Yaskawa INFORM job: DPRINT3D9.JBI

/JOB
//NAME DPRINT3D9
//POS
///NPOS 990,0,0,0,0,0
///TOOL 9
///POSTYPE PULSE
///PULSE
C00000=28405,51687,-122249,62656,-119296,-93988,0
C00001=28412,51716,-122153,62661,-119336,-93961,0
C00002=28422,51752,-122032,62666,-119387,-93929,0
C00003=28439,51788,-121908,62666,-119441,-93896,0
C00004=28474,51840,-121733,62650,-119521,-93851,0
C00005=28491,51862,-121660,62641,-119556,-93833,0
C00006=28516,51888,-121571,62626,-119598,-93812,0
C00007=28569,51934,-121420,62588,-119677,-93776,0
C00008=28598,51956,-121347,62567,-119716,-93759,0
C00009=28631,51978,-121273,62542,-119756,-93743,0
C00010=28686,52010,-121168,62495,-119817,-93721,0
C00011=28702,52019,-121138,62481,-119834,-93715,0
C00012=28783,52055,-121016,62410,-119911,-93692,0
C00013=28872,52087,-120913,62327,-119983,-93676,0
C00014=28965,52116,-120819,62238,-120053,-93663,0
C00015=29065,52138,-120745,62139,-120119,-93656,0
C00016=29167,52158,-120681,62036,-120181,-93653,0
C00017=29273,52171,-120639,61925,-120237,-93656,0
C00018=29381,52181,-120608,61811,-120288,-93663,0
C00019=29407,52182,-120605,61783,-120299,-93666,0
C00020=29496,52184,-120600,61686,-120334,-93678,0
C00021=29604,52182,-120611,61566,-120368,-93696,0
C00022=29681,52175,-120634,61479,-120388,-93714,0
C00023=29759,52166,-120666,61388,-120404,-93733,0
C00024=29816,52159,-120690,61322,-120414,-93748,0
C00025=29867,52150,-120721,61262,-120421,-93765,0
C00026=29912,52141,-120753,61208,-120425,-93780,0
C00027=30014,52117,-120835,61084,-120429,-93818,0
C00028=30081,52097,-120903,61002,-120426,-93846,0
C00029=30142,52075,-120975,60925,-120419,-93875,0
C00030=30190,52057,-121036,60863,-120412,-93899,0
C00031=30233,52039,-121099,60807,-120402,-93923,0
C00032=30261,52025,-121146,60769,-120394,-93940,0
C00033=30336,51984,-121284,60667,-120365,-93989,0
C00034=30393,51946,-121414,60587,-120333,-94033,0
C00035=30394,51945,-121416,60586,-120332,-94033,0
C00036=30454,51900,-121569,60498,-120291,-94084,0
C00037=25336,55338,-110610,67670,-122156,-90253,0
C00038=36363,52336,-120236,76454,-115258,-91971,0
C00039=39662,59274,-99499,75865,-122176,-86210,0
C00040=39594,59234,-99609,75915,-122109,-86232,0
C00041=39523,59198,-99708,75970,-122044,-86250,0
C00042=39446,59171,-99784,76034,-121979,-86261,0
C00043=39368,59147,-99848,76102,-121917,-86268,0
C00044=39340,59142,-99863,76127,-121898,-86268,0
C00045=39232,59125,-99908,76227,-121823,-86266,0
C00046=39175,59121,-99918,76282,-121786,-86261,0
C00047=39120,59120,-99919,76336,-121754,-86254,0
C00048=39037,59123,-99909,76421,-121707,-86239,0
C00049=38943,59135,-99873,76519,-121660,-86216,0
C00050=38887,59145,-99844,76580,-121634,-86200,0
C00051=38833,59159,-99805,76639,-121611,-86181,0
C00052=38779,59174,-99762,76699,-121589,-86161,0
C00053=38727,59193,-99708,76759,-121570,-86138,0
C00054=38679,59214,-99647,76815,-121557,-86114,0
C00055=38626,59240,-99574,76879,-121543,-86085,0
C00056=38582,59266,-99502,76934,-121534,-86059,0
C00057=38541,59294,-99421,76987,-121528,-86030,0
C00058=38493,59330,-99320,77050,-121522,-85994,0
C00059=38457,59362,-99230,77099,-121522,-85963,0
C00060=38425,59397,-99134,77146,-121524,-85931,0
C00061=38384,59443,-99005,77206,-121530,-85888,0
C00062=38358,59479,-98903,77248,-121537,-85855,0
C00063=38335,59518,-98796,77287,-121548,-85821,0
C00064=38305,59573,-98641,77340,-121566,-85773,0
C00065=38288,59612,-98533,77374,-121581,-85739,0
C00066=38275,59653,-98419,77404,-121599,-85704,0
C00067=38258,59716,-98245,77448,-121629,-85652,0
C00068=38251,59756,-98134,77472,-121650,-85619,0
C00069=38248,59798,-98018,77493,-121674,-85585,0
C00070=38246,59850,-97873,77518,-121706,-85543,0
C00071=38249,59905,-97721,77539,-121742,-85499,0
C00072=38262,59984,-97504,77560,-121800,-85439,0
C00073=38270,60017,-97413,77567,-121825,-85414,0
C00074=38282,60058,-97301,77572,-121858,-85383,0
C00075=38312,60130,-97103,77574,-121921,-85331,0
C00076=38328,60164,-97010,77573,-121953,-85306,0
C00077=38348,60200,-96910,77569,-121987,-85280,0
C00078=38384,60252,-96769,77557,-122041,-85245,0
C00079=38395,60266,-96729,77553,-122058,-85235,0
C00080=38449,60329,-96560,77528,-122129,-85194,0
C00081=38511,60384,-96409,77490,-122202,-85159,0
C00082=38578,60436,-96267,77449,-122276,-85127,0
C00083=38651,60480,-96148,77396,-122349,-85104,0
C00084=38728,60520,-96039,77339,-122421,-85083,0
C00085=38809,60551,-95956,77273,-122491,-85071,0
C00086=38893,60578,-95885,77204,-122560,-85063,0
C00087=38913,60582,-95874,77186,-122575,-85062,0
C00088=38984,60595,-95840,77122,-122628,-85063,0
C00089=39071,60603,-95818,77042,-122686,-85069,0
C00090=39134,60603,-95821,76980,-122725,-85079,0
C00091=39199,60598,-95835,76914,-122762,-85093,0
C00092=39246,60594,-95846,76866,-122790,-85102,0
C00093=39289,60587,-95867,76821,-122811,-85115,0
C00094=39328,60579,-95890,76779,-122830,-85127,0
C00095=39416,60556,-95955,76683,-122870,-85158,0
C00096=39474,60534,-96016,76616,-122892,-85184,0
C00097=39528,60510,-96084,76552,-122909,-85212,0
C00098=39571,60489,-96140,76500,-122923,-85234,0
C00099=39611,60467,-96203,76451,-122933,-85258,0
C00100=39637,60450,-96250,76418,-122938,-85275,0
C00101=39708,60399,-96390,76325,-122949,-85325,0
C00102=39763,60350,-96527,76249,-122950,-85373,0
C00103=39818,60293,-96684,76169,-122947,-85426,0
C00104=39841,60265,-96762,76134,-122942,-85451,0
C00105=39864,60231,-96854,76096,-122934,-85481,0
C00106=39908,60160,-97051,76020,-122915,-85544,0
C00107=39936,60100,-97217,75965,-122892,-85596,0
C00108=39963,60022,-97433,75902,-122856,-85661,0
C00109=39977,59961,-97602,75861,-122824,-85712,0
C00110=39985,59879,-97827,75816,-122775,-85777,0
C00111=39984,59819,-97993,75789,-122734,-85825,0
C00112=39974,59737,-98221,75762,-122672,-85888,0
C00113=39963,59689,-98351,75752,-122634,-85924,0
C00114=39939,59613,-98563,75741,-122569,-85981,0
C00115=39909,59548,-98742,75742,-122507,-86028,0
C00116=39874,59485,-98916,75748,-122445,-86073,0
C00117=39830,59427,-99078,75766,-122378,-86113,0
C00118=39781,59371,-99232,75789,-122312,-86150,0
C00119=39725,59322,-99367,75823,-122246,-86181,0
C00120=39667,59251,-99564,75850,-122163,-86229,0
C00121=39667,59198,-99585,75860,-122179,-86211,0
C00122=23846,60628,-95390,71835,-125896,-85715,0
C00123=23864,60580,-95520,71793,-125872,-85755,0
C00124=23881,60519,-95686,71745,-125836,-85803,0
C00125=23892,60475,-95806,71712,-125810,-85839,0
C00126=23898,60430,-95929,71683,-125780,-85875,0
C00127=23901,60372,-96089,71651,-125737,-85920,0
C00128=23902,60326,-96215,71627,-125704,-85955,0
C00129=23898,60280,-96341,71608,-125667,-85990,0
C00130=23888,60226,-96490,71590,-125620,-86030,0
C00131=23878,60180,-96615,71577,-125580,-86063,0
C00132=23863,60134,-96741,71569,-125536,-86096,0
C00133=23843,60086,-96871,71566,-125488,-86129,0
C00134=23822,60042,-96993,71565,-125443,-86159,0
C00135=23796,59999,-97111,71569,-125395,-86188,0
C00136=23767,59959,-97220,71578,-125348,-86214,0
C00137=23745,59929,-97302,71586,-125312,-86233,0
C00138=23696,59873,-97457,71608,-125240,-86268,0
C00139=23642,59819,-97604,71635,-125168,-86300,0
C00140=23581,59772,-97733,71674,-125096,-86326,0
C00141=23516,59729,-97852,71718,-125025,-86348,0
C00142=23445,59693,-97950,71772,-124957,-86364,0
C00143=23372,59661,-98036,71831,-124889,-86376,0
C00144=23294,59638,-98100,71898,-124826,-86381,0
C00145=23214,59619,-98150,71969,-124765,-86382,0
C00146=23133,59610,-98176,72047,-124711,-86376,0
C00147=23050,59605,-98189,72127,-124658,-86366,0
C00148=22968,59609,-98176,72212,-124613,-86349,0
C00149=22887,59618,-98151,72299,-124572,-86329,0
C00150=22807,59636,-98101,72388,-124539,-86301,0
C00151=22729,59658,-98038,72477,-124510,-86271,0
C00152=22656,59689,-97952,72566,-124489,-86235,0
C00153=22609,59711,-97889,72624,-124479,-86209,0
C00154=22517,59763,-97744,72742,-124462,-86154,0
C00155=22463,59801,-97639,72814,-124458,-86116,0
C00156=22396,59860,-97478,72909,-124460,-86059,0
C00157=22351,59907,-97347,72977,-124468,-86015,0
C00158=22299,59976,-97157,73063,-124487,-85953,0
C00159=22265,60032,-97002,73124,-124508,-85903,0
C00160=22230,60108,-96792,73196,-124542,-85839,0
C00161=22208,60171,-96619,73248,-124574,-85787,0
C00162=22192,60252,-96398,73303,-124621,-85722,0
C00163=22185,60319,-96213,73342,-124666,-85668,0
C00164=22187,60401,-95989,73380,-124726,-85605,0
C00165=22196,60471,-95799,73406,-124780,-85553,0
C00166=22216,60551,-95580,73425,-124849,-85495,0
C00167=22225,60580,-95500,73430,-124875,-85474,0
C00168=22239,60620,-95393,73434,-124912,-85446,0
C00169=22259,60660,-95284,73434,-124952,-85418,0
C00170=22285,60710,-95147,73433,-125004,-85384,0
C00171=22316,60760,-95011,73428,-125058,-85351,0
C00172=22368,60828,-94828,73409,-125137,-85308,0
C00173=22393,60857,-94749,73398,-125173,-85290,0
C00174=22424,60889,-94663,73383,-125214,-85271,0
C00175=22487,60943,-94515,73348,-125292,-85239,0
C00176=22520,60969,-94444,73328,-125332,-85225,0
C00177=22555,60994,-94377,73306,-125371,-85212,0
C00178=22579,61008,-94341,73288,-125395,-85206,0
C00179=22631,61034,-94269,73250,-125445,-85194,0
C00180=22709,61070,-94174,73190,-125519,-85181,0
C00181=22792,61096,-94105,73121,-125589,-85176,0
C00182=22876,61117,-94049,73048,-125656,-85174,0
C00183=22963,61127,-94021,72967,-125716,-85180,0
C00184=23030,61132,-94009,72903,-125761,-85188,0
C00185=23050,61133,-94006,72884,-125775,-85191,0
C00186=23137,61128,-94021,72795,-125826,-85210,0
C00187=23224,61119,-94048,72704,-125872,-85232,0
C00188=23265,61108,-94076,72658,-125890,-85247,0
C00189=23307,61096,-94111,72610,-125907,-85264,0
C00190=23389,61068,-94188,72514,-125937,-85300,0
C00191=23430,61049,-94240,72464,-125949,-85321,0
C00192=23465,61031,-94289,72420,-125958,-85341,0
C00193=23542,60986,-94410,72321,-125973,-85388,0
C00194=23591,60951,-94508,72254,-125977,-85424,0
C00195=23636,60913,-94611,72190,-125977,-85461,0
C00196=23671,60883,-94694,72140,-125976,-85490,0
C00197=23701,60851,-94779,72094,-125972,-85519,0
C00198=23722,60827,-94846,72060,-125967,-85541,0
C00199=23774,60760,-95028,71974,-125950,-85601,0
C00200=23805,60710,-95165,71918,-125931,-85644,0
C00201=23813,60696,-95204,71903,-125926,-85657,0
C00202=23853,60627,-95392,71827,-125899,-85717,0
C00203=35333,54219,-114032,78249,-116367,-89931,0
C00204=36296,54629,-112795,77405,-117135,-89659,0
C00205=40948,51484,-123021,71252,-116309,-93275,0
C00206=33829,55601,-109813,58647,-126335,-91484,0
C00207=35388,54173,-114177,78176,-116359,-89981,0
C00208=35604,54911,-111921,78224,-117000,-89320,0
C00209=36477,55304,-110751,77475,-117719,-89066,0
C00210=42176,51451,-123165,69910,-116723,-93454,0
C00211=33601,54921,-111852,58546,-125434,-91973,0
C00212=34232,54338,-113645,79428,-115921,-89701,0
C00213=35134,54709,-112527,78633,-116623,-89453,0
C00214=34899,54920,-111881,78950,-116654,-89233,0
C00215=35367,55123,-111276,78545,-117031,-89101,0
C00216=35550,54959,-111775,78297,-117007,-89271,0
C00217=36109,54680,-112634,77617,-117082,-89590,0
C00218=34833,55179,-111096,57314,-126251,-92011,0
C00219=36906,53447,-116478,54108,-124788,-93773,0
C00220=39302,53451,-116519,73803,-117568,-91120,0
C00221=44160,56039,-108728,69806,-122133,-89491,0
C00222=34853,55161,-111150,79086,-116797,-89008,0
C00223=32974,57094,-105422,81665,-116999,-87092,0
C00224=36073,54209,-114081,77479,-116712,-90024,0
C00225=40138,51461,-123080,72117,-115983,-93206,0
C00226=48458,53029,-118092,63773,-120900,-92785,0
C00227=48536,53068,-117968,63707,-120976,-92761,0
C00228=48617,53106,-117850,63636,-121052,-92741,0
C00229=48707,53137,-117753,63552,-121123,-92727,0
C00230=48778,53159,-117684,63485,-121176,-92718,0
C00231=48800,53165,-117664,63464,-121192,-92716,0
C00232=48899,53186,-117599,63366,-121257,-92712,0
C00233=49000,53205,-117541,63264,-121316,-92712,0
C00234=49051,53210,-117526,63211,-121343,-92714,0
C00235=49104,53214,-117515,63154,-121368,-92720,0
C00236=49210,53219,-117501,63041,-121415,-92732,0
C00237=49266,53219,-117503,62980,-121436,-92741,0
C00238=49315,53218,-117510,62925,-121453,-92750,0
C00239=49424,53211,-117533,62802,-121486,-92773,0
C00240=49498,53202,-117563,62717,-121505,-92793,0
C00241=49569,53191,-117601,62633,-121519,-92814,0
C00242=49625,53182,-117633,62568,-121528,-92831,0
C00243=49675,53170,-117671,62507,-121534,-92850,0
C00244=49713,53161,-117702,62461,-121536,-92864,0
C00245=49808,53133,-117794,62344,-121538,-92904,0
C00246=49870,53110,-117870,62264,-121534,-92935,0
C00247=49925,53086,-117947,62193,-121525,-92965,0
C00248=49970,53066,-118014,62133,-121517,-92989,0
C00249=50012,53044,-118087,62077,-121505,-93016,0
C00250=50065,53010,-118198,62002,-121483,-93055,0
C00251=50103,52985,-118280,61948,-121466,-93083,0
C00252=50136,52958,-118368,61899,-121445,-93113,0
C00253=50174,52921,-118487,61840,-121414,-93151,0
C00254=50202,52892,-118581,61795,-121388,-93182,0
C00255=50225,52862,-118681,61755,-121358,-93213,0
C00256=50247,52824,-118803,61714,-121319,-93250,0
C00257=50264,52793,-118907,61680,-121285,-93281,0
C00258=50275,52759,-119016,61651,-121247,-93313,0
C00259=50281,52723,-119133,61627,-121204,-93346,0
C00260=50286,52689,-119243,61606,-121162,-93378,0
C00261=50284,52655,-119356,61592,-121119,-93408,0
C00262=50277,52622,-119464,61584,-121073,-93437,0
C00263=50271,52597,-119546,61579,-121039,-93459,0
C00264=50252,52547,-119708,61576,-120969,-93501,0
C00265=50226,52499,-119866,61582,-120898,-93541,0
C00266=50188,52452,-120018,61601,-120825,-93578,0
C00267=50145,52407,-120166,61628,-120751,-93612,0
C00268=50089,52365,-120302,61669,-120677,-93642,0
C00269=50029,52325,-120432,61718,-120604,-93670,0
C00270=49958,52290,-120548,61779,-120533,-93692,0
C00271=49882,52257,-120656,61846,-120464,-93711,0
C00272=49799,52229,-120746,61926,-120398,-93724,0
C00273=49711,52203,-120828,62010,-120334,-93734,0
C00274=49618,52184,-120890,62104,-120276,-93738,0
C00275=49523,52168,-120942,62201,-120221,-93739,0
C00276=49424,52158,-120973,62305,-120174,-93733,0
C00277=49324,52151,-120992,62412,-120130,-93725,0
C00278=49223,52150,-120991,62523,-120094,-93710,0
C00279=49157,52152,-120984,62596,-120073,-93699,0
C00280=49023,52159,-120954,62748,-120035,-93672,0
C00281=48939,52169,-120922,62844,-120018,-93651,0
C00282=48829,52187,-120858,62974,-120002,-93617,0
C00283=48749,52204,-120798,63070,-119996,-93589,0
C00284=48649,52233,-120699,63193,-119996,-93547,0
C00285=48576,52259,-120613,63285,-120003,-93512,0
C00286=48491,52297,-120484,63396,-120019,-93464,0
C00287=48429,52330,-120373,63479,-120038,-93424,0
C00288=48362,52376,-120220,63574,-120071,-93371,0
C00289=48313,52416,-120087,63646,-120103,-93327,0
C00290=48267,52467,-119916,63721,-120149,-93271,0
C00291=48235,52512,-119766,63777,-120194,-93224,0
C00292=48210,52568,-119583,63830,-120251,-93169,0
C00293=48203,52589,-119516,63848,-120274,-93149,0
C00294=48196,52617,-119421,63868,-120306,-93122,0
C00295=48194,52647,-119323,63884,-120343,-93093,0
C00296=48194,52686,-119197,63903,-120389,-93058,0
C00297=48198,52726,-119067,63916,-120438,-93022,0
C00298=48218,52782,-118884,63921,-120514,-92973,0
C00299=48229,52807,-118803,63920,-120549,-92952,0
C00300=48245,52836,-118711,63917,-120588,-92928,0
C00301=48283,52888,-118545,63898,-120665,-92887,0
C00302=48305,52913,-118462,63886,-120704,-92866,0
C00303=48333,52941,-118372,63869,-120748,-92845,0
C00304=48395,52987,-118225,63823,-120827,-92813,0
C00305=48451,53041,-118053,63787,-120912,-92772,0
C00306=39639,59169,-99665,75875,-122143,-86229,0
C00307=39576,59139,-99746,75925,-122086,-86244,0
C00308=39529,59119,-99801,75962,-122045,-86253,0
C00309=39481,59103,-99847,76003,-122006,-86259,0
C00310=39416,59085,-99893,76060,-121955,-86263,0
C00311=39364,59073,-99927,76106,-121917,-86266,0
C00312=39311,59064,-99950,76155,-121881,-86265,0
C00313=39248,59058,-99966,76216,-121839,-86260,0
C00314=39193,59054,-99975,76269,-121805,-86255,0
C00315=39137,59055,-99973,76324,-121771,-86247,0
C00316=39078,59059,-99960,76385,-121740,-86235,0
C00317=39022,59064,-99944,76443,-121711,-86222,0
C00318=38967,59074,-99916,76503,-121684,-86207,0
C00319=38914,59087,-99879,76561,-121662,-86189,0
C00320=38874,59097,-99849,76605,-121645,-86175,0
C00321=38797,59122,-99778,76692,-121616,-86143,0
C00322=38722,59152,-99694,76779,-121591,-86109,0
C00323=38652,59189,-99589,76864,-121575,-86069,0
C00324=38586,59230,-99474,76948,-121562,-86027,0
C00325=38527,59278,-99340,77027,-121558,-85980,0
C00326=38472,59329,-99197,77103,-121559,-85931,0
C00327=38426,59386,-99038,77173,-121567,-85879,0
C00328=38385,59445,-98873,77239,-121581,-85826,0
C00329=38353,59509,-98695,77298,-121602,-85770,0
C00330=38326,59574,-98514,77352,-121628,-85714,0
C00331=38311,59642,-98325,77397,-121661,-85657,0
C00332=38300,59711,-98134,77438,-121699,-85601,0
C00333=38300,59781,-97941,77468,-121743,-85545,0
C00334=38306,59851,-97748,77492,-121790,-85491,0
C00335=38322,59920,-97558,77507,-121844,-85438,0
C00336=38335,59964,-97436,77513,-121879,-85405,0
C00337=38370,60055,-97187,77518,-121958,-85338,0
C00338=38398,60110,-97036,77514,-122009,-85299,0
C00339=38446,60182,-96838,77499,-122084,-85249,0
C00340=38487,60233,-96699,77481,-122140,-85214,0
C00341=38550,60296,-96527,77448,-122218,-85174,0
C00342=38603,60341,-96406,77416,-122279,-85147,0
C00343=38677,60392,-96267,77365,-122357,-85118,0
C00344=38741,60428,-96169,77320,-122420,-85098,0
C00345=38824,60465,-96070,77254,-122494,-85082,0
C00346=38896,60491,-96001,77196,-122554,-85072,0
C00347=38986,60513,-95942,77118,-122624,-85068,0
C00348=39063,60526,-95908,77048,-122680,-85069,0
C00349=39155,60532,-95892,76961,-122741,-85078,0
C00350=39189,60533,-95891,76928,-122763,-85083,0
C00351=39236,60532,-95894,76882,-122791,-85090,0
C00352=39284,60527,-95909,76833,-122818,-85102,0
C00353=39345,60520,-95930,76770,-122852,-85117,0
C00354=39408,60508,-95963,76704,-122883,-85135,0
C00355=39495,60483,-96033,76607,-122921,-85168,0
C00356=39533,60470,-96069,76564,-122936,-85184,0
C00357=39575,60454,-96116,76514,-122952,-85203,0
C00358=39652,60416,-96221,76422,-122973,-85245,0
C00359=39689,60395,-96278,76377,-122984,-85267,0
C00360=39725,60372,-96341,76331,-122991,-85290,0
C00361=39746,60356,-96387,76302,-122993,-85306,0
C00362=39790,60320,-96487,76243,-122996,-85341,0
C00363=39850,60263,-96644,76158,-122996,-85394,0
C00364=39901,60200,-96818,76079,-122986,-85452,0
C00365=39948,60135,-96998,76004,-122972,-85510,0
C00366=39984,60064,-97192,75936,-122947,-85571,0
C00367=40015,59992,-97391,75872,-122918,-85632,0
C00368=40035,59918,-97597,75819,-122882,-85694,0
C00369=40049,59842,-97805,75770,-122839,-85756,0
C00370=40049,59786,-97962,75745,-122801,-85801,0
C00371=40041,59689,-98229,75709,-122732,-85876,0
C00372=40028,59634,-98380,75697,-122687,-85917,0
C00373=40010,59581,-98527,75690,-122641,-85957,0
C00374=39997,59541,-98637,75686,-122606,-85986,0
C00375=39980,59506,-98735,75687,-122572,-86012,0
C00376=39963,59476,-98816,75690,-122543,-86033,0
C00377=39920,59407,-99008,75702,-122469,-86081,0
C00378=39883,59362,-99132,75718,-122417,-86112,0
C00379=39845,59321,-99244,75738,-122368,-86138,0
C00380=39813,59289,-99333,75756,-122326,-86159,0
C00381=39778,59260,-99414,75777,-122286,-86177,0
C00382=39721,59219,-99527,75816,-122225,-86202,0
C00383=39708,59210,-99551,75825,-122212,-86207,0
C00384=39637,59145,-99731,75867,-122125,-86248,0
C00385=29173,52068,-120796,62026,-120175,-93660,0
C00386=29284,52085,-120742,61912,-120237,-93660,0
C00387=29377,52096,-120708,61815,-120284,-93664,0
C00388=29491,52102,-120690,61692,-120334,-93675,0
C00389=29589,52104,-120687,61586,-120371,-93689,0
C00390=29703,52099,-120703,61458,-120405,-93710,0
C00391=29744,52097,-120713,61411,-120417,-93719,0
C00392=29801,52091,-120731,61346,-120430,-93732,0
C00393=29859,52083,-120759,61279,-120440,-93748,0
C00394=29932,52073,-120796,61193,-120452,-93769,0
C00395=30005,52059,-120842,61106,-120460,-93793,0
C00396=30106,52034,-120928,60983,-120463,-93831,0
C00397=30150,52022,-120969,60930,-120461,-93848,0
C00398=30198,52006,-121021,60869,-120458,-93870,0
C00399=30283,51974,-121132,60760,-120444,-93913,0
C00400=30324,51956,-121191,60707,-120435,-93935,0
C00401=30363,51938,-121253,60655,-120425,-93958,0
C00402=30386,51925,-121298,60624,-120414,-93974,0
C00403=30430,51896,-121394,60562,-120391,-94007,0
C00404=30491,51853,-121542,60474,-120353,-94057,0
C00405=30540,51806,-121700,60398,-120306,-94107,0
C00406=30582,51757,-121863,60329,-120255,-94159,0
C00407=30610,51707,-122035,60274,-120195,-94210,0
C00408=30632,51656,-122207,60227,-120133,-94261,0
C00409=30639,51604,-122383,60195,-120063,-94310,0
C00410=30639,51552,-122559,60171,-119991,-94359,0
C00411=30626,51514,-122688,60168,-119934,-94393,0
C00412=30593,51451,-122906,60174,-119833,-94448,0
C00413=30564,51415,-123026,60190,-119774,-94478,0
C00414=30530,51381,-123142,60212,-119714,-94505,0
C00415=30503,51356,-123229,60230,-119670,-94525,0
C00416=30474,51334,-123304,60252,-119629,-94542,0
C00417=30447,51316,-123366,60274,-119595,-94556,0
C00418=30376,51273,-123511,60332,-119511,-94586,0
C00419=30320,51246,-123602,60382,-119455,-94604,0
C00420=30264,51223,-123682,60434,-119403,-94619,0
C00421=30216,51204,-123747,60477,-119360,-94630,0
C00422=30166,51188,-123802,60525,-119321,-94639,0
C00423=30086,51165,-123878,60604,-119264,-94649,0
C00424=30030,51151,-123927,60659,-119225,-94655,0
C00425=29972,51139,-123967,60717,-119189,-94658,0
C00426=29887,51125,-124015,60805,-119142,-94660,0
C00427=29825,51116,-124046,60869,-119108,-94661,0
C00428=29761,51109,-124067,60937,-119078,-94658,0
C00429=29677,51103,-124086,61027,-119042,-94652,0
C00430=29611,51100,-124097,61099,-119016,-94647,0
C00431=29544,51099,-124100,61172,-118992,-94638,0
C00432=29464,51100,-124093,61261,-118969,-94625,0
C00433=29396,51103,-124084,61337,-118949,-94614,0
C00434=29327,51108,-124064,61415,-118934,-94599,0
C00435=29256,51116,-124034,61498,-118922,-94581,0
C00436=29189,51125,-124003,61576,-118912,-94563,0
C00437=29123,51136,-123962,61654,-118907,-94543,0
C00438=29062,51149,-123915,61727,-118904,-94521,0
C00439=29015,51160,-123877,61783,-118904,-94505,0
C00440=28927,51184,-123793,61891,-118908,-94469,0
C00441=28843,51210,-123700,61996,-118916,-94431,0
C00442=28768,51241,-123589,62093,-118933,-94390,0
C00443=28697,51275,-123473,62186,-118956,-94348,0
C00444=28637,51313,-123342,62270,-118986,-94303,0
C00445=28583,51352,-123206,62347,-119021,-94257,0
C00446=28540,51394,-123060,62413,-119064,-94209,0
C00447=28504,51438,-122909,62472,-119111,-94162,0
C00448=28482,51484,-122752,62518,-119164,-94114,0
C00449=28466,51531,-122593,62557,-119220,-94067,0
C00450=28463,51578,-122431,62581,-119282,-94021,0
C00451=28467,51626,-122270,62599,-119347,-93976,0
C00452=28484,51673,-122110,62601,-119414,-93933,0
C00453=28508,51719,-121953,62596,-119485,-93892,0
C00454=28544,51764,-121802,62577,-119556,-93854,0
C00455=28571,51793,-121706,62560,-119603,-93830,0
C00456=28635,51851,-121512,62517,-119701,-93784,0
C00457=28682,51886,-121397,62481,-119763,-93759,0
C00458=28758,51930,-121250,62419,-119848,-93728,0
C00459=28819,51961,-121149,62365,-119909,-93708,0
C00460=28910,51997,-121028,62282,-119989,-93687,0
C00461=28985,52023,-120945,62211,-120049,-93674,0
C00462=29079,52048,-120864,62120,-120114,-93665,0
C00463=29175,52074,-120779,62026,-120183,-93655,0
C00464=25374,55292,-110598,67645,-122208,-90230,0
C00465=36364,52274,-120259,76461,-115276,-91949,0
C00466=36364,52212,-120281,76469,-115296,-91927,0
C00467=23335,59560,-98191,71855,-124849,-86390,0
C00468=23306,59553,-98210,71882,-124827,-86390,0
C00469=23213,59536,-98255,71967,-124759,-86387,0
C00470=23136,59530,-98272,72041,-124710,-86380,0
C00471=23041,59529,-98274,72137,-124653,-86364,0
C00472=22966,59535,-98255,72216,-124614,-86347,0
C00473=22872,59550,-98212,72318,-124571,-86319,0
C00474=22802,59569,-98161,72397,-124543,-86293,0
C00475=22713,59600,-98073,72502,-124513,-86254,0
C00476=22651,59629,-97993,72578,-124498,-86221,0
C00477=22571,59675,-97864,72681,-124485,-86172,0
C00478=22527,59706,-97779,72740,-124482,-86141,0
C00479=22459,59760,-97628,72835,-124481,-86087,0
C00480=22406,59813,-97481,72914,-124488,-86037,0
C00481=22356,59869,-97326,72991,-124500,-85986,0
C00482=22342,59891,-97268,73015,-124506,-85967,0
C00483=22293,59973,-97042,73104,-124536,-85895,0
C00484=22272,60018,-96918,73146,-124557,-85857,0
C00485=22256,60062,-96796,73184,-124579,-85820,0
C00486=22236,60131,-96607,73237,-124616,-85763,0
C00487=22226,60202,-96412,73281,-124662,-85707,0
C00488=22222,60273,-96217,73320,-124710,-85651,0
C00489=22229,60345,-96021,73348,-124764,-85597,0
C00490=22236,60392,-95894,73364,-124802,-85563,0
C00491=22248,60440,-95761,73376,-124843,-85527,0
C00492=22280,60531,-95515,73388,-124927,-85463,0
C00493=22289,60554,-95452,73390,-124949,-85447,0
C00494=22326,60619,-95275,73385,-125018,-85403,0
C00495=22367,60681,-95105,73375,-125087,-85362,0
C00496=22422,60747,-94928,73352,-125167,-85321,0
C00497=22459,60786,-94821,73336,-125217,-85297,0
C00498=22526,60847,-94656,73299,-125302,-85262,0
C00499=22580,60888,-94547,73265,-125364,-85240,0
C00500=22658,60935,-94420,73211,-125445,-85217,0
C00501=22721,60966,-94336,73165,-125506,-85205,0
C00502=22807,60999,-94249,73095,-125582,-85195,0
C00503=22877,61019,-94196,73036,-125639,-85191,0
C00504=22927,61028,-94171,72991,-125677,-85192,0
C00505=22993,61038,-94143,72931,-125726,-85196,0
C00506=23042,61043,-94132,72884,-125759,-85201,0
C00507=23092,61043,-94132,72834,-125790,-85210,0
C00508=23163,61041,-94137,72764,-125833,-85223,0
C00509=23210,61037,-94150,72714,-125859,-85235,0
C00510=23259,61028,-94174,72662,-125883,-85250,0
C00511=23331,61013,-94215,72582,-125916,-85274,0
C00512=23375,61001,-94250,72532,-125935,-85291,0
C00513=23421,60984,-94296,72478,-125951,-85312,0
C00514=23476,60962,-94356,72412,-125969,-85338,0
C00515=23531,60935,-94429,72343,-125984,-85368,0
C00516=23607,60889,-94555,72245,-125997,-85416,0
C00517=23637,60868,-94612,72204,-126000,-85438,0
C00518=23674,60841,-94688,72153,-126003,-85465,0
C00519=23735,60785,-94840,72064,-125999,-85519,0
C00520=23763,60757,-94917,72022,-125996,-85545,0
C00521=23792,60725,-95004,71977,-125990,-85574,0
C00522=23834,60667,-95161,71905,-125973,-85625,0
C00523=23880,60589,-95375,71819,-125943,-85693,0
C00524=23910,60514,-95578,71752,-125906,-85755,0
C00525=23934,60439,-95784,71689,-125865,-85817,0
C00526=23947,60361,-95997,71638,-125814,-85878,0
C00527=23954,60283,-96210,71591,-125760,-85939,0
C00528=23949,60205,-96423,71556,-125698,-85998,0
C00529=23939,60128,-96635,71527,-125635,-86055,0
C00530=23917,60053,-96841,71512,-125565,-86109,0
C00531=23906,60022,-96926,71508,-125534,-86131,0
C00532=23887,59980,-97041,71506,-125491,-86160,0
C00533=23867,59944,-97139,71508,-125452,-86184,0
C00534=23846,59911,-97228,71513,-125415,-86206,0
C00535=23799,59847,-97406,71528,-125338,-86247,0
C00536=23770,59813,-97498,71541,-125296,-86268,0
C00537=23744,59787,-97569,71554,-125261,-86283,0
C00538=23680,59729,-97728,71590,-125180,-86318,0
C00539=23631,59694,-97826,71622,-125124,-86336,0
C00540=23580,59662,-97912,71658,-125069,-86352,0
C00541=23540,59638,-97978,71687,-125028,-86364,0
C00542=23498,59618,-98033,71719,-124988,-86372,0
C00543=23468,59605,-98068,71743,-124960,-86377,0
C00544=23414,59585,-98123,71787,-124914,-86384,0
C00545=23328,59535,-98260,71850,-124826,-86408,0
C00546=35333,54161,-114054,78257,-116384,-89910,0
C00547=36296,54570,-112817,77413,-117151,-89638,0
C00548=40948,51421,-123044,71260,-116332,-93253,0
C00549=33830,55544,-109834,58658,-126362,-91466,0
C00550=35388,54114,-114198,78183,-116376,-89960,0
C00551=35604,54853,-111943,78232,-117016,-89300,0
C00552=36477,55247,-110773,77483,-117736,-89046,0
C00553=42176,51388,-123187,69918,-116747,-93432,0
C00554=33601,54863,-111874,58557,-125460,-91955,0
C00555=34233,54280,-113666,79435,-115937,-89680,0
C00556=35134,54651,-112549,78640,-116639,-89432,0
C00557=34899,54862,-111903,78958,-116670,-89213,0
C00558=35368,55065,-111298,78553,-117047,-89080,0
C00559=35550,54901,-111797,78305,-117023,-89250,0
C00560=36110,54622,-112655,77625,-117098,-89570,0
C00561=34833,55122,-111117,57326,-126280,-91993,0
C00562=36892,53399,-116465,54141,-124829,-93744,0
C00563=39302,53391,-116540,73812,-117587,-91099,0
C00564=44131,55963,-108806,69839,-122123,-89484,0
C00565=34853,55104,-111172,79094,-116813,-88987,0
C00566=32987,57025,-105483,81656,-117012,-87085,0
C00567=36073,54150,-114102,77487,-116729,-90003,0
C00568=40138,51398,-123103,72125,-116006,-93184,0
C00569=48644,53016,-117967,63603,-121053,-92751,0
C00570=48694,53036,-117903,63558,-121097,-92741,0
C00571=48760,53061,-117824,63497,-121152,-92728,0
C00572=48813,53078,-117772,63448,-121192,-92722,0
C00573=48868,53092,-117729,63394,-121230,-92718,0
C00574=48946,53111,-117670,63317,-121283,-92713,0
C00575=49002,53122,-117637,63261,-121316,-92712,0
C00576=49060,53130,-117613,63202,-121349,-92714,0
C00577=49148,53141,-117579,63111,-121396,-92718,0
C00578=49204,53146,-117566,63051,-121423,-92723,0
C00579=49263,53148,-117561,62988,-121449,-92731,0
C00580=49336,53150,-117557,62909,-121478,-92741,0
C00581=49412,53149,-117562,62824,-121506,-92754,0
C00582=49521,53141,-117591,62701,-121538,-92778,0
C00583=49567,53136,-117607,62649,-121551,-92789,0
C00584=49623,53129,-117631,62584,-121562,-92805,0
C00585=49722,53111,-117692,62467,-121578,-92837,0
C00586=49768,53101,-117725,62411,-121584,-92853,0
C00587=49818,53088,-117767,62350,-121588,-92872,0
C00588=49898,53064,-117847,62251,-121588,-92907,0
C00589=49994,53027,-117969,62128,-121578,-92955,0
C00590=50069,52987,-118096,62026,-121559,-93002,0
C00591=50140,52946,-118232,61929,-121535,-93050,0
C00592=50199,52900,-118381,61841,-121499,-93101,0
C00593=50254,52852,-118538,61759,-121460,-93152,0
C00594=50295,52801,-118703,61689,-121412,-93204,0
C00595=50331,52749,-118873,61625,-121359,-93256,0
C00596=50352,52695,-119050,61575,-121299,-93308,0
C00597=50358,52672,-119125,61558,-121272,-93330,0
C00598=50363,52640,-119228,61537,-121234,-93359,0
C00599=50363,52612,-119320,61524,-121198,-93385,0
C00600=50360,52585,-119408,61514,-121162,-93408,0
C00601=50349,52531,-119583,61501,-121090,-93455,0
C00602=50337,52502,-119679,61500,-121047,-93480,0
C00603=50325,52478,-119757,61502,-121013,-93500,0
C00604=50291,52424,-119934,61514,-120931,-93544,0
C00605=50259,52388,-120051,61532,-120874,-93571,0
C00606=50224,52354,-120160,61555,-120818,-93596,0
C00607=50194,52328,-120246,61575,-120774,-93616,0
C00608=50161,52304,-120326,61600,-120730,-93633,0
C00609=50136,52288,-120379,61620,-120700,-93644,0
C00610=50062,52244,-120520,61681,-120619,-93673,0
C00611=49991,52211,-120627,61744,-120551,-93692,0
C00612=49901,52176,-120743,61827,-120473,-93711,0
C00613=49820,52151,-120823,61905,-120412,-93722,0
C00614=49716,52124,-120907,62007,-120342,-93730,0
C00615=49629,52108,-120958,62095,-120290,-93732,0
C00616=49516,52093,-121007,62212,-120230,-93730,0
C00617=49428,52085,-121029,62307,-120190,-93724,0
C00618=49309,52081,-121039,62435,-120143,-93710,0
C00619=49223,52082,-121033,62531,-120114,-93696,0
C00620=49105,52090,-121005,62664,-120082,-93671,0
C00621=49037,52097,-120979,62742,-120067,-93654,0
C00622=48928,52113,-120923,62869,-120049,-93623,0
C00623=48835,52132,-120858,62980,-120040,-93592,0
C00624=48746,52153,-120784,63088,-120035,-93558,0
C00625=48717,52163,-120752,63124,-120037,-93545,0
C00626=48612,52200,-120625,63257,-120047,-93494,0
C00627=48561,52223,-120549,63323,-120057,-93466,0
C00628=48516,52246,-120471,63383,-120070,-93437,0
C00629=48452,52283,-120345,63471,-120093,-93393,0
C00630=48399,52325,-120207,63549,-120125,-93346,0
C00631=48351,52368,-120064,63621,-120160,-93299,0
C00632=48315,52414,-119910,63682,-120204,-93251,0
C00633=48296,52445,-119808,63718,-120235,-93219,0
C00634=48280,52479,-119698,63751,-120271,-93186,0
C00635=48262,52544,-119485,63800,-120343,-93122,0
C00636=48259,52561,-119428,63811,-120363,-93106,0
C00637=48262,52612,-119264,63832,-120425,-93060,0
C00638=48271,52662,-119100,63845,-120489,-93015,0
C00639=48295,52718,-118918,63845,-120566,-92967,0
C00640=48312,52753,-118807,63842,-120613,-92938,0
C00641=48352,52810,-118622,63825,-120697,-92892,0
C00642=48389,52850,-118493,63804,-120759,-92861,0
C00643=48449,52902,-118327,63763,-120843,-92824,0
C00644=48500,52939,-118210,63724,-120907,-92798,0
C00645=48570,52979,-118083,63667,-120982,-92772,0
C00646=48641,53022,-117947,63609,-121060,-92745,0
C00647=30481,51730,-121766,60467,-120297,-94091,0
C00648=30492,51720,-121799,60451,-120288,-94102,0
C00649=30519,51690,-121899,60406,-120257,-94133,0
C00650=30540,51662,-121997,60370,-120225,-94163,0
C00651=30565,51624,-122125,60325,-120181,-94202,0
C00652=30578,51595,-122224,60297,-120145,-94231,0
C00653=30586,51565,-122324,60274,-120107,-94260,0
C00654=30595,51523,-122466,60245,-120052,-94301,0
C00655=30596,51495,-122562,60230,-120013,-94328,0
C00656=30591,51466,-122661,60222,-119972,-94354,0
C00657=30582,51422,-122809,60212,-119907,-94394,0
C00658=30571,51395,-122902,60212,-119866,-94418,0
C00659=30554,51367,-122996,60217,-119821,-94442,0
C00660=30532,51334,-123111,60226,-119767,-94471,0
C00661=30503,51299,-123230,60242,-119709,-94499,0
C00662=30450,51252,-123391,60280,-119625,-94537,0
C00663=30425,51232,-123457,60298,-119588,-94552,0
C00664=30391,51209,-123538,60325,-119544,-94570,0
C00665=30321,51169,-123672,60384,-119465,-94597,0
C00666=30285,51151,-123734,60415,-119428,-94610,0
C00667=30244,51132,-123799,60453,-119388,-94622,0
C00668=30168,51103,-123896,60524,-119323,-94639,0
C00669=30062,51071,-124007,60626,-119242,-94655,0
C00670=29959,51049,-124081,60729,-119177,-94662,0
C00671=29854,51030,-124147,60837,-119116,-94666,0
C00672=29744,51017,-124188,60953,-119062,-94663,0
C00673=29632,51007,-124220,61072,-119011,-94657,0
C00674=29518,51004,-124228,61196,-118970,-94644,0
C00675=29404,51005,-124225,61322,-118933,-94628,0
C00676=29292,51012,-124198,61449,-118907,-94606,0
C00677=29246,51016,-124181,61502,-118897,-94594,0
C00678=29182,51024,-124155,61576,-118887,-94579,0
C00679=29128,51032,-124123,61640,-118881,-94562,0
C00680=29078,51042,-124088,61699,-118878,-94546,0
C00681=28977,51064,-124011,61820,-118876,-94510,0
C00682=28925,51078,-123961,61884,-118878,-94489,0
C00683=28884,51091,-123915,61935,-118882,-94471,0
C00684=28793,51123,-123802,62050,-118895,-94427,0
C00685=28735,51148,-123713,62125,-118911,-94394,0
C00686=28684,51175,-123623,62194,-118930,-94361,0
C00687=28644,51196,-123548,62247,-118944,-94335,0
C00688=28610,51218,-123471,62295,-118963,-94309,0
C00689=28588,51234,-123416,62326,-118978,-94290,0
C00690=28532,51281,-123255,62409,-119021,-94237,0
C00691=28495,51322,-123111,62468,-119065,-94191,0
C00692=28460,51374,-122936,62529,-119121,-94137,0
C00693=28443,51417,-122786,62569,-119174,-94092,0
C00694=28431,51472,-122601,62606,-119242,-94038,0
C00695=28432,51515,-122454,62624,-119300,-93996,0
C00696=28445,51570,-122267,62636,-119377,-93945,0
C00697=28463,51612,-122127,62634,-119437,-93908,0
C00698=28499,51666,-121945,62620,-119520,-93862,0
C00699=28533,51704,-121817,62600,-119582,-93830,0
C00700=28591,51755,-121648,62560,-119668,-93790,0
C00701=28630,51783,-121555,62530,-119719,-93769,0
C00702=28699,51827,-121407,62473,-119802,-93738,0
C00703=28769,51863,-121289,62414,-119873,-93714,0
C00704=28816,51885,-121215,62372,-119919,-93700,0
C00705=28842,51897,-121177,62349,-119943,-93693,0
C00706=28924,51926,-121082,62272,-120010,-93678,0
C00707=29010,51952,-120996,62190,-120074,-93666,0
C00708=29041,51960,-120972,62160,-120095,-93664,0
C00709=29101,51973,-120928,62100,-120134,-93660,0
C00710=29195,51991,-120869,62005,-120191,-93657,0
C00711=29293,52003,-120830,61903,-120242,-93660,0
C00712=29392,52012,-120803,61798,-120289,-93667,0
C00713=29492,52015,-120795,61689,-120329,-93679,0
C00714=29593,52015,-120798,61579,-120365,-93694,0
C00715=29692,52008,-120822,61466,-120391,-93715,0
C00716=29790,51998,-120857,61354,-120413,-93739,0
C00717=29823,51993,-120874,61315,-120418,-93749,0
C00718=29885,51982,-120911,61242,-120426,-93768,0
C00719=29977,51964,-120975,61131,-120434,-93799,0
C00720=30075,51937,-121066,61011,-120434,-93838,0
C00721=30135,51919,-121128,60936,-120430,-93865,0
C00722=30190,51899,-121196,60867,-120423,-93891,0
C00723=30243,51878,-121265,60798,-120414,-93918,0
C00724=30293,51855,-121342,60733,-120402,-93946,0
C00725=30337,51832,-121422,60673,-120384,-93975,0
C00726=30385,51804,-121515,60608,-120365,-94008,0
C00727=30430,51773,-121620,60544,-120338,-94043,0
C00728=30505,51730,-121767,60441,-120305,-94094,0
C00729=25413,55246,-110586,67621,-122259,-90207,0
C00730=36364,52212,-120281,76469,-115296,-91927,0
C00731=39711,59118,-99680,75815,-122204,-86220,0
C00732=39637,59075,-99799,75870,-122130,-86243,0
C00733=39559,59036,-99906,75930,-122058,-86262,0
C00734=39475,59006,-99989,76000,-121989,-86275,0
C00735=39390,58980,-100060,76074,-121921,-86283,0
C00736=39301,58963,-100103,76155,-121858,-86282,0
C00737=39210,58952,-100134,76240,-121797,-86279,0
C00738=39119,58950,-100136,76330,-121743,-86267,0
C00739=39081,58952,-100131,76369,-121722,-86260,0
C00740=39028,58956,-100119,76423,-121693,-86249,0
C00741=38982,58963,-100098,76472,-121671,-86236,0
C00742=38940,58972,-100074,76518,-121652,-86224,0
C00743=38854,58993,-100013,76613,-121615,-86194,0
C00744=38808,59008,-99970,76665,-121598,-86175,0
C00745=38772,59022,-99929,76707,-121586,-86159,0
C00746=38689,59059,-99826,76805,-121561,-86117,0
C00747=38636,59089,-99740,76871,-121550,-86085,0
C00748=38587,59121,-99649,76933,-121542,-86052,0
C00749=38549,59148,-99574,76982,-121537,-86026,0
C00750=38515,59176,-99495,77028,-121535,-85998,0
C00751=38493,59197,-99436,77059,-121535,-85978,0
C00752=38434,59258,-99265,77143,-121539,-85921,0
C00753=38393,59314,-99108,77208,-121551,-85870,0
C00754=38350,59385,-98913,77280,-121570,-85808,0
C00755=38323,59446,-98743,77333,-121593,-85755,0
C00756=38298,59523,-98530,77391,-121627,-85690,0
C00757=38286,59585,-98356,77430,-121660,-85638,0
C00758=38280,59666,-98133,77471,-121706,-85573,0
C00759=38283,59728,-97961,77494,-121747,-85524,0
C00760=38296,59810,-97736,77517,-121807,-85462,0
C00761=38313,59869,-97575,77526,-121853,-85417,0
C00762=38344,59948,-97358,77530,-121922,-85359,0
C00763=38368,59992,-97235,77526,-121964,-85327,0
C00764=38411,60064,-97039,77515,-122036,-85277,0
C00765=38456,60123,-96877,77497,-122100,-85237,0
C00766=38506,60180,-96721,77473,-122167,-85199,0
C00767=38563,60231,-96583,77439,-122233,-85167,0
C00768=38624,60279,-96453,77401,-122301,-85139,0
C00769=38692,60320,-96344,77353,-122368,-85117,0
C00770=38762,60356,-96244,77300,-122434,-85098,0
C00771=38837,60385,-96168,77240,-122499,-85087,0
C00772=38914,60409,-96103,77176,-122562,-85080,0
C00773=38993,60424,-96063,77105,-122621,-85079,0
C00774=39073,60435,-96035,77031,-122677,-85083,0
C00775=39154,60437,-96032,76953,-122729,-85094,0
C00776=39236,60434,-96042,76872,-122777,-85109,0
C00777=39263,60430,-96053,76844,-122791,-85116,0
C00778=39315,60421,-96077,76789,-122818,-85130,0
C00779=39394,60405,-96125,76704,-122856,-85155,0
C00780=39480,60377,-96203,76608,-122891,-85190,0
C00781=39532,60357,-96257,76547,-122911,-85213,0
C00782=39581,60334,-96320,76490,-122926,-85238,0
C00783=39629,60310,-96387,76431,-122941,-85264,0
C00784=39675,60283,-96463,76374,-122952,-85293,0
C00785=39716,60253,-96545,76320,-122957,-85322,0
C00786=39761,60219,-96640,76260,-122963,-85356,0
C00787=39802,60182,-96741,76204,-122964,-85391,0
C00788=39819,60163,-96794,76177,-122962,-85409,0
C00789=39869,60109,-96945,76104,-122956,-85459,0
C00790=39899,60069,-97055,76056,-122949,-85495,0
C00791=39923,60029,-97165,76014,-122938,-85530,0
C00792=39953,59976,-97310,75961,-122921,-85576,0
C00793=39972,59936,-97422,75924,-122906,-85611,0
C00794=39986,59894,-97538,75890,-122886,-85646,0
C00795=40005,59834,-97703,75845,-122857,-85696,0
C00796=40014,59793,-97817,75817,-122836,-85730,0
C00797=40018,59750,-97936,75794,-122810,-85765,0
C00798=40023,59685,-98114,75760,-122769,-85816,0
C00799=40022,59645,-98226,75742,-122741,-85848,0
C00800=40016,59602,-98342,75729,-122710,-85880,0
C00801=40008,59551,-98485,75713,-122670,-85920,0
C00802=39995,59497,-98633,75702,-122626,-85960,0
C00803=39966,59422,-98840,75697,-122560,-86015,0
C00804=39952,59391,-98926,75697,-122530,-86038,0
C00805=39932,59354,-99030,75701,-122492,-86065,0
C00806=39888,59289,-99209,75715,-122422,-86110,0
C00807=39865,59258,-99293,75725,-122389,-86131,0
C00808=39837,59226,-99382,75738,-122351,-86152,0
C00809=39785,59177,-99519,75767,-122286,-86184,0
C00810=39774,59167,-99547,75774,-122272,-86190,0
C00811=39714,59101,-99727,75804,-122193,-86233,0
C00812=39715,59048,-99748,75814,-122209,-86215,0
C00813=23644,60735,-94855,72168,-125962,-85483,0
C00814=23666,60715,-94908,72136,-125961,-85502,0
C00815=23696,60688,-94982,72092,-125959,-85528,0
C00816=23732,60649,-95089,72036,-125953,-85564,0
C00817=23785,60579,-95280,71948,-125934,-85626,0
C00818=23822,60520,-95441,71881,-125913,-85678,0
C00819=23857,60447,-95641,71809,-125880,-85740,0
C00820=23879,60385,-95809,71755,-125847,-85790,0
C00821=23899,60304,-96032,71695,-125799,-85856,0
C00822=23908,60238,-96211,71653,-125756,-85908,0
C00823=23909,60156,-96437,71610,-125693,-85971,0
C00824=23903,60088,-96621,71583,-125639,-86022,0
C00825=23885,60008,-96841,71560,-125569,-86080,0
C00826=23864,59942,-97022,71548,-125506,-86127,0
C00827=23828,59867,-97228,71546,-125428,-86178,0
C00828=23814,59840,-97301,71548,-125399,-86196,0
C00829=23792,59804,-97400,71552,-125359,-86220,0
C00830=23764,59769,-97497,71562,-125317,-86243,0
C00831=23729,59724,-97618,71576,-125261,-86271,0
C00832=23688,59681,-97737,71595,-125205,-86297,0
C00833=23622,59625,-97891,71634,-125124,-86329,0
C00834=23592,59601,-97956,71654,-125088,-86343,0
C00835=23554,59576,-98026,71679,-125047,-86356,0
C00836=23480,59534,-98140,71734,-124972,-86376,0
C00837=23442,59515,-98193,71763,-124935,-86384,0
C00838=23401,59497,-98242,71795,-124897,-86391,0
C00839=23366,59485,-98273,71825,-124868,-86394,0
C00840=23317,59471,-98312,71868,-124828,-86396,0
C00841=23230,59450,-98368,71945,-124762,-86398,0
C00842=23141,59440,-98395,72030,-124702,-86391,0
C00843=23051,59434,-98410,72118,-124645,-86380,0
C00844=22961,59439,-98396,72211,-124596,-86361,0
C00845=22872,59448,-98369,72305,-124551,-86339,0
C00846=22785,59468,-98313,72402,-124514,-86309,0
C00847=22719,59487,-98261,72478,-124489,-86284,0
C00848=22700,59492,-98245,72500,-124482,-86276,0
C00849=22665,59507,-98205,72542,-124473,-86260,0
C00850=22621,59528,-98146,72597,-124463,-86236,0
C00851=22543,59571,-98026,72696,-124448,-86189,0
C00852=22494,59606,-97930,72762,-124444,-86154,0
C00853=22447,59644,-97824,72828,-124444,-86117,0
C00854=22412,59673,-97744,72876,-124446,-86088,0
C00855=22384,59702,-97662,72919,-124450,-86061,0
C00856=22360,59729,-97589,72956,-124456,-86036,0
C00857=22309,59795,-97407,73039,-124472,-85977,0
C00858=22279,59844,-97271,73092,-124490,-85934,0
C00859=22255,59892,-97139,73140,-124511,-85892,0
C00860=22236,59932,-97029,73178,-124528,-85859,0
C00861=22222,59972,-96920,73211,-124548,-85826,0
C00862=22206,60035,-96746,73257,-124585,-85774,0
C00863=22197,60078,-96627,73287,-124610,-85739,0
C00864=22192,60122,-96509,73313,-124637,-85705,0
C00865=22191,60184,-96339,73344,-124681,-85657,0
C00866=22192,60229,-96216,73365,-124713,-85622,0
C00867=22197,60273,-96094,73382,-124748,-85589,0
C00868=22209,60331,-95936,73398,-124796,-85546,0
C00869=22220,60377,-95813,73409,-124835,-85513,0
C00870=22236,60422,-95691,73415,-124876,-85481,0
C00871=22259,60473,-95551,73417,-124927,-85446,0
C00872=22280,60517,-95432,73418,-124971,-85416,0
C00873=22305,60559,-95317,73413,-125017,-85387,0
C00874=22337,60603,-95198,73403,-125066,-85360,0
C00875=22368,60643,-95089,73392,-125114,-85334,0
C00876=22403,60681,-94985,73376,-125163,-85310,0
C00877=22441,60716,-94891,73356,-125210,-85290,0
C00878=22481,60751,-94797,73333,-125259,-85270,0
C00879=22532,60789,-94693,73302,-125318,-85249,0
C00880=22596,60834,-94573,73260,-125389,-85227,0
C00881=22666,60871,-94475,73209,-125458,-85210,0
C00882=22738,60903,-94388,73154,-125525,-85198,0
C00883=22814,60927,-94324,73090,-125589,-85193,0
C00884=22891,60946,-94273,73023,-125650,-85192,0
C00885=22971,60956,-94247,72949,-125706,-85198,0
C00886=23023,60960,-94238,72899,-125742,-85204,0
C00887=23051,60961,-94234,72872,-125760,-85208,0
C00888=23131,60957,-94247,72791,-125806,-85225,0
C00889=23210,60948,-94272,72707,-125849,-85246,0
C00890=23288,60929,-94323,72621,-125883,-85273,0
C00891=23338,60914,-94364,72564,-125904,-85293,0
C00892=23388,60896,-94415,72504,-125922,-85316,0
C00893=23482,60851,-94536,72389,-125947,-85366,0
C00894=23506,60839,-94571,72358,-125952,-85380,0
C00895=23583,60785,-94718,72254,-125961,-85434,0
C00896=23673,60743,-94833,72142,-125985,-85482,0
C00897=35334,54102,-114076,78265,-116400,-89889,0
C00898=36296,54512,-112838,77421,-117168,-89618,0
C00899=40949,51358,-123065,71268,-116355,-93231,0
C00900=33830,55487,-109856,58670,-126389,-91449,0
C00901=35388,54056,-114220,78191,-116392,-89938,0
C00902=35604,54795,-111965,78240,-117032,-89279,0
C00903=36477,55190,-110794,77492,-117753,-89026,0
C00904=42176,51325,-123210,69926,-116771,-93410,0
C00905=33602,54806,-111896,58568,-125488,-91937,0
C00906=34233,54221,-113688,79443,-115953,-89658,0
C00907=35135,54593,-112570,78648,-116655,-89412,0
C00908=34900,54804,-111924,78966,-116686,-89192,0
C00909=35368,55008,-111319,78561,-117063,-89059,0
C00910=35550,54843,-111818,78313,-117039,-89229,0
C00911=36110,54564,-112677,77633,-117115,-89549,0
C00912=34834,55064,-111139,57337,-126307,-91975,0
C00913=36877,53350,-116452,54174,-124870,-93715,0
C00914=39302,53332,-116562,73820,-117607,-91078,0
C00915=44101,55888,-108883,69872,-122112,-89475,0
C00916=34853,55046,-111193,79101,-116829,-88966,0
C00917=32999,56956,-105544,81647,-117024,-87078,0
C00918=36073,54091,-114124,77495,-116746,-89982,0
C00919=40138,51335,-123125,72133,-116028,-93162,0
C00920=48321,52700,-118802,63847,-120653,-92912,0
C00921=48362,52747,-118651,63824,-120725,-92876,0
C00922=48407,52793,-118504,63796,-120797,-92841,0
C00923=48464,52836,-118369,63754,-120868,-92811,0
C00924=48526,52876,-118240,63706,-120941,-92784,0
C00925=48596,52913,-118125,63645,-121011,-92763,0
C00926=48671,52947,-118018,63579,-121080,-92743,0
C00927=48754,52975,-117929,63503,-121145,-92731,0
C00928=48839,53001,-117847,63421,-121208,-92721,0
C00929=48930,53021,-117786,63332,-121267,-92717,0
C00930=49022,53038,-117734,63238,-121323,-92717,0
C00931=49118,53048,-117705,63138,-121372,-92723,0
C00932=49215,53055,-117685,63035,-121417,-92732,0
C00933=49312,53056,-117686,62929,-121455,-92748,0
C00934=49409,53053,-117698,62821,-121489,-92765,0
C00935=49505,53043,-117732,62712,-121514,-92789,0
C00936=49599,53030,-117776,62603,-121534,-92815,0
C00937=49621,53026,-117791,62576,-121537,-92823,0
C00938=49656,53020,-117810,62535,-121543,-92834,0
C00939=49704,53011,-117840,62478,-121551,-92850,0
C00940=49766,52996,-117890,62402,-121557,-92873,0
C00941=49865,52967,-117986,62280,-121558,-92915,0
C00942=49940,52939,-118077,62185,-121552,-92951,0
C00943=50021,52902,-118196,62078,-121537,-92996,0
C00944=50081,52869,-118304,61996,-121520,-93036,0
C00945=50150,52823,-118456,61898,-121488,-93088,0
C00946=50199,52783,-118585,61825,-121457,-93131,0
C00947=50249,52731,-118756,61745,-121409,-93186,0
C00948=50283,52686,-118901,61687,-121367,-93231,0
C00949=50312,52630,-119084,61628,-121307,-93286,0
C00950=50329,52582,-119241,61586,-121252,-93332,0
C00951=50336,52524,-119428,61551,-121182,-93385,0
C00952=50336,52503,-119496,61541,-121155,-93404,0
C00953=50334,52474,-119591,61529,-121118,-93429,0
C00954=50326,52444,-119689,61524,-121076,-93455,0
C00955=50315,52406,-119813,61519,-121023,-93488,0
C00956=50297,52368,-119939,61520,-120968,-93520,0
C00957=50260,52314,-120114,61535,-120887,-93563,0
C00958=50242,52291,-120190,61545,-120850,-93581,0
C00959=50217,52264,-120276,61560,-120807,-93602,0
C00960=50161,52218,-120428,61599,-120727,-93636,0
C00961=50131,52195,-120502,61621,-120688,-93652,0
C00962=50098,52173,-120574,61647,-120648,-93667,0
C00963=50067,52156,-120629,61674,-120614,-93678,0
C00964=50022,52134,-120702,61713,-120569,-93692,0
C00965=49940,52097,-120820,61787,-120494,-93712,0
C00966=49848,52067,-120919,61873,-120421,-93726,0
C00967=49753,52039,-121007,61965,-120352,-93738,0
C00968=49651,52018,-121075,62068,-120289,-93742,0
C00969=49547,52000,-121132,62174,-120229,-93743,0
C00970=49439,51989,-121165,62288,-120178,-93737,0
C00971=49355,51983,-121183,62378,-120140,-93730,0
C00972=49330,51982,-121188,62405,-120129,-93728,0
C00973=49282,51981,-121188,62457,-120112,-93721,0
C00974=49220,51982,-121181,62526,-120093,-93710,0
C00975=49106,51989,-121158,62654,-120060,-93688,0
C00976=49030,51997,-121128,62742,-120044,-93668,0
C00977=48954,52008,-121089,62831,-120032,-93647,0
C00978=48898,52017,-121058,62897,-120022,-93630,0
C00979=48847,52028,-121020,62957,-120018,-93613,0
C00980=48805,52038,-120985,63008,-120017,-93597,0
C00981=48707,52065,-120892,63129,-120016,-93557,0
C00982=48644,52088,-120815,63209,-120021,-93526,0
C00983=48587,52111,-120736,63282,-120030,-93496,0
C00984=48542,52131,-120669,63341,-120038,-93471,0
C00985=48502,52152,-120599,63394,-120051,-93445,0
C00986=48446,52187,-120482,63472,-120074,-93404,0
C00987=48409,52211,-120400,63523,-120091,-93376,0
C00988=48378,52237,-120315,63570,-120111,-93347,0
C00989=48339,52275,-120189,63630,-120144,-93306,0
//INST
///DATE 2025/02/20 16:20
///COMM Generated using RoboDK
///ATTR SC,RW
///GROUP1 RB1
NOP
MOVL C00000 V=30.0 PL=1
MOVL C00001 V=30.0 PL=1
MOVL C00002 V=30.0 PL=1
MOVL C00003 V=30.0 PL=1
MOVL C00004 V=30.0 PL=1
MOVL C00005 V=30.0 PL=1
MOVL C00006 V=30.0 PL=1
MOVL C00007 V=30.0 PL=1
MOVL C00008 V=30.0 PL=1
MOVL C00009 V=30.0 PL=1
MOVL C00010 V=30.0 PL=1
MOVL C00011 V=30.0 PL=1
MOVL C00012 V=30.0 PL=1
MOVL C00013 V=30.0 PL=1
MOVL C00014 V=30.0 PL=1
MOVL C00015 V=30.0 PL=1
MOVL C00016 V=30.0 PL=1
MOVL C00017 V=30.0 PL=1
MOVL C00018 V=30.0 PL=1
MOVL C00019 V=30.0 PL=1
MOVL C00020 V=30.0 PL=1
MOVL C00021 V=30.0 PL=1
MOVL C00022 V=30.0 PL=1
MOVL C00023 V=30.0 PL=1
MOVL C00024 V=30.0 PL=1
MOVL C00025 V=30.0 PL=1
MOVL C00026 V=30.0 PL=1
MOVL C00027 V=30.0 PL=1
MOVL C00028 V=30.0 PL=1
MOVL C00029 V=30.0 PL=1
MOVL C00030 V=30.0 PL=1
MOVL C00031 V=30.0 PL=1
MOVL C00032 V=30.0 PL=1
MOVL C00033 V=30.0 PL=1
MOVL C00034 V=30.0 PL=1
MOVL C00035 V=30.0 PL=1
MOVL C00036 V=130.0 PL=1
MOVL C00037 V=130.0 PL=1
MOVL C00038 V=30.0 PL=1
MOVL C00039 V=130.0 PL=1
MOVL C00040 V=30.0 PL=1
MOVL C00041 V=30.0 PL=1
MOVL C00042 V=30.0 PL=1
MOVL C00043 V=30.0 PL=1
MOVL C00044 V=30.0 PL=1
MOVL C00045 V=30.0 PL=1
MOVL C00046 V=30.0 PL=1
MOVL C00047 V=30.0 PL=1
MOVL C00048 V=30.0 PL=1
MOVL C00049 V=30.0 PL=1
MOVL C00050 V=30.0 PL=1
MOVL C00051 V=30.0 PL=1
MOVL C00052 V=30.0 PL=1
MOVL C00053 V=30.0 PL=1
MOVL C00054 V=30.0 PL=1
MOVL C00055 V=30.0 PL=1
MOVL C00056 V=30.0 PL=1
MOVL C00057 V=30.0 PL=1
MOVL C00058 V=30.0 PL=1
MOVL C00059 V=30.0 PL=1
MOVL C00060 V=30.0 PL=1
MOVL C00061 V=30.0 PL=1
MOVL C00062 V=30.0 PL=1
MOVL C00063 V=30.0 PL=1
MOVL C00064 V=30.0 PL=1
MOVL C00065 V=30.0 PL=1
MOVL C00066 V=30.0 PL=1
MOVL C00067 V=30.0 PL=1
MOVL C00068 V=30.0 PL=1
MOVL C00069 V=30.0 PL=1
MOVL C00070 V=30.0 PL=1
MOVL C00071 V=30.0 PL=1
MOVL C00072 V=30.0 PL=1
MOVL C00073 V=30.0 PL=1
MOVL C00074 V=30.0 PL=1
MOVL C00075 V=30.0 PL=1
MOVL C00076 V=30.0 PL=1
MOVL C00077 V=30.0 PL=1
MOVL C00078 V=30.0 PL=1
MOVL C00079 V=30.0 PL=1
MOVL C00080 V=30.0 PL=1
MOVL C00081 V=30.0 PL=1
MOVL C00082 V=30.0 PL=1
MOVL C00083 V=30.0 PL=1
MOVL C00084 V=30.0 PL=1
MOVL C00085 V=30.0 PL=1
MOVL C00086 V=30.0 PL=1
MOVL C00087 V=30.0 PL=1
MOVL C00088 V=30.0 PL=1
MOVL C00089 V=30.0 PL=1
MOVL C00090 V=30.0 PL=1
MOVL C00091 V=30.0 PL=1
MOVL C00092 V=30.0 PL=1
MOVL C00093 V=30.0 PL=1
MOVL C00094 V=30.0 PL=1
MOVL C00095 V=30.0 PL=1
MOVL C00096 V=30.0 PL=1
MOVL C00097 V=30.0 PL=1
MOVL C00098 V=30.0 PL=1
MOVL C00099 V=30.0 PL=1
MOVL C00100 V=30.0 PL=1
MOVL C00101 V=30.0 PL=1
MOVL C00102 V=30.0 PL=1
MOVL C00103 V=30.0 PL=1
MOVL C00104 V=30.0 PL=1
MOVL C00105 V=30.0 PL=1
MOVL C00106 V=30.0 PL=1
MOVL C00107 V=30.0 PL=1
MOVL C00108 V=30.0 PL=1
MOVL C00109 V=30.0 PL=1
MOVL C00110 V=30.0 PL=1
MOVL C00111 V=30.0 PL=1
MOVL C00112 V=30.0 PL=1
MOVL C00113 V=30.0 PL=1
MOVL C00114 V=30.0 PL=1
MOVL C00115 V=30.0 PL=1
MOVL C00116 V=30.0 PL=1
MOVL C00117 V=30.0 PL=1
MOVL C00118 V=30.0 PL=1
MOVL C00119 V=30.0 PL=1
MOVL C00120 V=130.0 PL=1
MOVL C00121 V=130.0 PL=1
MOVL C00122 V=130.0 PL=1
MOVL C00123 V=30.0 PL=1
MOVL C00124 V=30.0 PL=1
MOVL C00125 V=30.0 PL=1
MOVL C00126 V=30.0 PL=1
MOVL C00127 V=30.0 PL=1
MOVL C00128 V=30.0 PL=1
MOVL C00129 V=30.0 PL=1
MOVL C00130 V=30.0 PL=1
MOVL C00131 V=30.0 PL=1
MOVL C00132 V=30.0 PL=1
MOVL C00133 V=30.0 PL=1
MOVL C00134 V=30.0 PL=1
MOVL C00135 V=30.0 PL=1
MOVL C00136 V=30.0 PL=1
MOVL C00137 V=30.0 PL=1
MOVL C00138 V=30.0 PL=1
MOVL C00139 V=30.0 PL=1
MOVL C00140 V=30.0 PL=1
MOVL C00141 V=30.0 PL=1
MOVL C00142 V=30.0 PL=1
MOVL C00143 V=30.0 PL=1
MOVL C00144 V=30.0 PL=1
MOVL C00145 V=30.0 PL=1
MOVL C00146 V=30.0 PL=1
MOVL C00147 V=30.0 PL=1
MOVL C00148 V=30.0 PL=1
MOVL C00149 V=30.0 PL=1
MOVL C00150 V=30.0 PL=1
MOVL C00151 V=30.0 PL=1
MOVL C00152 V=30.0 PL=1
MOVL C00153 V=30.0 PL=1
MOVL C00154 V=30.0 PL=1
MOVL C00155 V=30.0 PL=1
MOVL C00156 V=30.0 PL=1
MOVL C00157 V=30.0 PL=1
MOVL C00158 V=30.0 PL=1
MOVL C00159 V=30.0 PL=1
MOVL C00160 V=30.0 PL=1
MOVL C00161 V=30.0 PL=1
MOVL C00162 V=30.0 PL=1
MOVL C00163 V=30.0 PL=1
MOVL C00164 V=30.0 PL=1
MOVL C00165 V=30.0 PL=1
MOVL C00166 V=30.0 PL=1
MOVL C00167 V=30.0 PL=1
MOVL C00168 V=30.0 PL=1
MOVL C00169 V=30.0 PL=1
MOVL C00170 V=30.0 PL=1
MOVL C00171 V=30.0 PL=1
MOVL C00172 V=30.0 PL=1
MOVL C00173 V=30.0 PL=1
MOVL C00174 V=30.0 PL=1
MOVL C00175 V=30.0 PL=1
MOVL C00176 V=30.0 PL=1
MOVL C00177 V=30.0 PL=1
MOVL C00178 V=30.0 PL=1
MOVL C00179 V=30.0 PL=1
MOVL C00180 V=30.0 PL=1
MOVL C00181 V=30.0 PL=1
MOVL C00182 V=30.0 PL=1
MOVL C00183 V=30.0 PL=1
MOVL C00184 V=30.0 PL=1
MOVL C00185 V=30.0 PL=1
MOVL C00186 V=30.0 PL=1
MOVL C00187 V=30.0 PL=1
MOVL C00188 V=30.0 PL=1
MOVL C00189 V=30.0 PL=1
MOVL C00190 V=30.0 PL=1
MOVL C00191 V=30.0 PL=1
MOVL C00192 V=30.0 PL=1
MOVL C00193 V=30.0 PL=1
MOVL C00194 V=30.0 PL=1
MOVL C00195 V=30.0 PL=1
MOVL C00196 V=30.0 PL=1
MOVL C00197 V=30.0 PL=1
MOVL C00198 V=30.0 PL=1
MOVL C00199 V=30.0 PL=1
MOVL C00200 V=30.0 PL=1
MOVL C00201 V=30.0 PL=1
MOVL C00202 V=130.0 PL=1
MOVL C00203 V=130.0 PL=1
MOVL C00204 V=60.0 PL=1
MOVL C00205 V=60.0 PL=1
MOVL C00206 V=60.0 PL=1
MOVL C00207 V=60.0 PL=1
MOVL C00208 V=130.0 PL=1
MOVL C00209 V=30.0 PL=1
MOVL C00210 V=30.0 PL=1
MOVL C00211 V=30.0 PL=1
MOVL C00212 V=30.0 PL=1
MOVL C00213 V=30.0 PL=1
MOVL C00214 V=30.0 PL=1
MOVL C00215 V=30.0 PL=1
MOVL C00216 V=30.0 PL=1
MOVL C00217 V=130.0 PL=1
MOVL C00218 V=130.0 PL=1
MOVL C00219 V=30.0 PL=1
MOVL C00220 V=130.0 PL=1
MOVL C00221 V=30.0 PL=1
MOVL C00222 V=130.0 PL=1
MOVL C00223 V=30.0 PL=1
MOVL C00224 V=130.0 PL=1
MOVL C00225 V=20.0 PL=1
MOVL C00226 V=130.0 PL=1
MOVL C00227 V=30.0 PL=1
MOVL C00228 V=30.0 PL=1
MOVL C00229 V=30.0 PL=1
MOVL C00230 V=30.0 PL=1
MOVL C00231 V=30.0 PL=1
MOVL C00232 V=30.0 PL=1
MOVL C00233 V=30.0 PL=1
MOVL C00234 V=30.0 PL=1
MOVL C00235 V=30.0 PL=1
MOVL C00236 V=30.0 PL=1
MOVL C00237 V=30.0 PL=1
MOVL C00238 V=30.0 PL=1
MOVL C00239 V=30.0 PL=1
MOVL C00240 V=30.0 PL=1
MOVL C00241 V=30.0 PL=1
MOVL C00242 V=30.0 PL=1
MOVL C00243 V=30.0 PL=1
MOVL C00244 V=30.0 PL=1
MOVL C00245 V=30.0 PL=1
MOVL C00246 V=30.0 PL=1
MOVL C00247 V=30.0 PL=1
MOVL C00248 V=30.0 PL=1
MOVL C00249 V=30.0 PL=1
MOVL C00250 V=30.0 PL=1
MOVL C00251 V=30.0 PL=1
MOVL C00252 V=30.0 PL=1
MOVL C00253 V=30.0 PL=1
MOVL C00254 V=30.0 PL=1
MOVL C00255 V=30.0 PL=1
MOVL C00256 V=30.0 PL=1
MOVL C00257 V=30.0 PL=1
MOVL C00258 V=30.0 PL=1
MOVL C00259 V=30.0 PL=1
MOVL C00260 V=30.0 PL=1
MOVL C00261 V=30.0 PL=1
MOVL C00262 V=30.0 PL=1
MOVL C00263 V=30.0 PL=1
MOVL C00264 V=30.0 PL=1
MOVL C00265 V=30.0 PL=1
MOVL C00266 V=30.0 PL=1
MOVL C00267 V=30.0 PL=1
MOVL C00268 V=30.0 PL=1
MOVL C00269 V=30.0 PL=1
MOVL C00270 V=30.0 PL=1
MOVL C00271 V=30.0 PL=1
MOVL C00272 V=30.0 PL=1
MOVL C00273 V=30.0 PL=1
MOVL C00274 V=30.0 PL=1
MOVL C00275 V=30.0 PL=1
MOVL C00276 V=30.0 PL=1
MOVL C00277 V=30.0 PL=1
MOVL C00278 V=30.0 PL=1
MOVL C00279 V=30.0 PL=1
MOVL C00280 V=30.0 PL=1
MOVL C00281 V=30.0 PL=1
MOVL C00282 V=30.0 PL=1
MOVL C00283 V=30.0 PL=1
MOVL C00284 V=30.0 PL=1
MOVL C00285 V=30.0 PL=1
MOVL C00286 V=30.0 PL=1
MOVL C00287 V=30.0 PL=1
MOVL C00288 V=30.0 PL=1
MOVL C00289 V=30.0 PL=1
MOVL C00290 V=30.0 PL=1
MOVL C00291 V=30.0 PL=1
MOVL C00292 V=30.0 PL=1
MOVL C00293 V=30.0 PL=1
MOVL C00294 V=30.0 PL=1
MOVL C00295 V=30.0 PL=1
MOVL C00296 V=30.0 PL=1
MOVL C00297 V=30.0 PL=1
MOVL C00298 V=30.0 PL=1
MOVL C00299 V=30.0 PL=1
MOVL C00300 V=30.0 PL=1
MOVL C00301 V=30.0 PL=1
MOVL C00302 V=30.0 PL=1
MOVL C00303 V=30.0 PL=1
MOVL C00304 V=30.0 PL=1
MOVL C00305 V=130.0 PL=1
MOVL C00306 V=130.0 PL=1
MOVL C00307 V=30.0 PL=1
MOVL C00308 V=30.0 PL=1
MOVL C00309 V=30.0 PL=1
MOVL C00310 V=30.0 PL=1
MOVL C00311 V=30.0 PL=1
MOVL C00312 V=30.0 PL=1
MOVL C00313 V=30.0 PL=1
MOVL C00314 V=30.0 PL=1
MOVL C00315 V=30.0 PL=1
MOVL C00316 V=30.0 PL=1
MOVL C00317 V=30.0 PL=1
MOVL C00318 V=30.0 PL=1
MOVL C00319 V=30.0 PL=1
MOVL C00320 V=30.0 PL=1
MOVL C00321 V=30.0 PL=1
MOVL C00322 V=30.0 PL=1
MOVL C00323 V=30.0 PL=1
MOVL C00324 V=30.0 PL=1
MOVL C00325 V=30.0 PL=1
MOVL C00326 V=30.0 PL=1
MOVL C00327 V=30.0 PL=1
MOVL C00328 V=30.0 PL=1
MOVL C00329 V=30.0 PL=1
MOVL C00330 V=30.0 PL=1
MOVL C00331 V=30.0 PL=1
MOVL C00332 V=30.0 PL=1
MOVL C00333 V=30.0 PL=1
MOVL C00334 V=30.0 PL=1
MOVL C00335 V=30.0 PL=1
MOVL C00336 V=30.0 PL=1
MOVL C00337 V=30.0 PL=1
MOVL C00338 V=30.0 PL=1
MOVL C00339 V=30.0 PL=1
MOVL C00340 V=30.0 PL=1
MOVL C00341 V=30.0 PL=1
MOVL C00342 V=30.0 PL=1
MOVL C00343 V=30.0 PL=1
MOVL C00344 V=30.0 PL=1
MOVL C00345 V=30.0 PL=1
MOVL C00346 V=30.0 PL=1
MOVL C00347 V=30.0 PL=1
MOVL C00348 V=30.0 PL=1
MOVL C00349 V=30.0 PL=1
MOVL C00350 V=30.0 PL=1
MOVL C00351 V=30.0 PL=1
MOVL C00352 V=30.0 PL=1
MOVL C00353 V=30.0 PL=1
MOVL C00354 V=30.0 PL=1
MOVL C00355 V=30.0 PL=1
MOVL C00356 V=30.0 PL=1
MOVL C00357 V=30.0 PL=1
MOVL C00358 V=30.0 PL=1
MOVL C00359 V=30.0 PL=1
MOVL C00360 V=30.0 PL=1
MOVL C00361 V=30.0 PL=1
MOVL C00362 V=30.0 PL=1
MOVL C00363 V=30.0 PL=1
MOVL C00364 V=30.0 PL=1
MOVL C00365 V=30.0 PL=1
MOVL C00366 V=30.0 PL=1
MOVL C00367 V=30.0 PL=1
MOVL C00368 V=30.0 PL=1
MOVL C00369 V=30.0 PL=1
MOVL C00370 V=30.0 PL=1
MOVL C00371 V=30.0 PL=1
MOVL C00372 V=30.0 PL=1
MOVL C00373 V=30.0 PL=1
MOVL C00374 V=30.0 PL=1
MOVL C00375 V=30.0 PL=1
MOVL C00376 V=30.0 PL=1
MOVL C00377 V=30.0 PL=1
MOVL C00378 V=30.0 PL=1
MOVL C00379 V=30.0 PL=1
MOVL C00380 V=30.0 PL=1
MOVL C00381 V=30.0 PL=1
MOVL C00382 V=30.0 PL=1
MOVL C00383 V=30.0 PL=1
MOVL C00384 V=130.0 PL=1
MOVL C00385 V=130.0 PL=1
MOVL C00386 V=30.0 PL=1
MOVL C00387 V=30.0 PL=1
MOVL C00388 V=30.0 PL=1
MOVL C00389 V=30.0 PL=1
MOVL C00390 V=30.0 PL=1
MOVL C00391 V=30.0 PL=1
MOVL C00392 V=30.0 PL=1
MOVL C00393 V=30.0 PL=1
MOVL C00394 V=30.0 PL=1
MOVL C00395 V=30.0 PL=1
MOVL C00396 V=30.0 PL=1
MOVL C00397 V=30.0 PL=1
MOVL C00398 V=30.0 PL=1
MOVL C00399 V=30.0 PL=1
MOVL C00400 V=30.0 PL=1
MOVL C00401 V=30.0 PL=1
MOVL C00402 V=30.0 PL=1
MOVL C00403 V=30.0 PL=1
MOVL C00404 V=30.0 PL=1
MOVL C00405 V=30.0 PL=1
MOVL C00406 V=30.0 PL=1
MOVL C00407 V=30.0 PL=1
MOVL C00408 V=30.0 PL=1
MOVL C00409 V=30.0 PL=1
MOVL C00410 V=30.0 PL=1
MOVL C00411 V=30.0 PL=1
MOVL C00412 V=30.0 PL=1
MOVL C00413 V=30.0 PL=1
MOVL C00414 V=30.0 PL=1
MOVL C00415 V=30.0 PL=1
MOVL C00416 V=30.0 PL=1
MOVL C00417 V=30.0 PL=1
MOVL C00418 V=30.0 PL=1
MOVL C00419 V=30.0 PL=1
MOVL C00420 V=30.0 PL=1
MOVL C00421 V=30.0 PL=1
MOVL C00422 V=30.0 PL=1
MOVL C00423 V=30.0 PL=1
MOVL C00424 V=30.0 PL=1
MOVL C00425 V=30.0 PL=1
MOVL C00426 V=30.0 PL=1
MOVL C00427 V=30.0 PL=1
MOVL C00428 V=30.0 PL=1
MOVL C00429 V=30.0 PL=1
MOVL C00430 V=30.0 PL=1
MOVL C00431 V=30.0 PL=1
MOVL C00432 V=30.0 PL=1
MOVL C00433 V=30.0 PL=1
MOVL C00434 V=30.0 PL=1
MOVL C00435 V=30.0 PL=1
MOVL C00436 V=30.0 PL=1
MOVL C00437 V=30.0 PL=1
MOVL C00438 V=30.0 PL=1
MOVL C00439 V=30.0 PL=1
MOVL C00440 V=30.0 PL=1
MOVL C00441 V=30.0 PL=1
MOVL C00442 V=30.0 PL=1
MOVL C00443 V=30.0 PL=1
MOVL C00444 V=30.0 PL=1
MOVL C00445 V=30.0 PL=1
MOVL C00446 V=30.0 PL=1
MOVL C00447 V=30.0 PL=1
MOVL C00448 V=30.0 PL=1
MOVL C00449 V=30.0 PL=1
MOVL C00450 V=30.0 PL=1
MOVL C00451 V=30.0 PL=1
MOVL C00452 V=30.0 PL=1
MOVL C00453 V=30.0 PL=1
MOVL C00454 V=30.0 PL=1
MOVL C00455 V=30.0 PL=1
MOVL C00456 V=30.0 PL=1
MOVL C00457 V=30.0 PL=1
MOVL C00458 V=30.0 PL=1
MOVL C00459 V=30.0 PL=1
MOVL C00460 V=30.0 PL=1
MOVL C00461 V=30.0 PL=1
MOVL C00462 V=30.0 PL=1
MOVL C00463 V=130.0 PL=1
MOVL C00464 V=130.0 PL=1
MOVL C00465 V=30.0 PL=1
MOVL C00466 V=130.0 PL=1
MOVL C00467 V=130.0 PL=1
MOVL C00468 V=30.0 PL=1
MOVL C00469 V=30.0 PL=1
MOVL C00470 V=30.0 PL=1
MOVL C00471 V=30.0 PL=1
MOVL C00472 V=30.0 PL=1
MOVL C00473 V=30.0 PL=1
MOVL C00474 V=30.0 PL=1
MOVL C00475 V=30.0 PL=1
MOVL C00476 V=30.0 PL=1
MOVL C00477 V=30.0 PL=1
MOVL C00478 V=30.0 PL=1
MOVL C00479 V=30.0 PL=1
MOVL C00480 V=30.0 PL=1
MOVL C00481 V=30.0 PL=1
MOVL C00482 V=30.0 PL=1
MOVL C00483 V=30.0 PL=1
MOVL C00484 V=30.0 PL=1
MOVL C00485 V=30.0 PL=1
MOVL C00486 V=30.0 PL=1
MOVL C00487 V=30.0 PL=1
MOVL C00488 V=30.0 PL=1
MOVL C00489 V=30.0 PL=1
MOVL C00490 V=30.0 PL=1
MOVL C00491 V=30.0 PL=1
MOVL C00492 V=30.0 PL=1
MOVL C00493 V=30.0 PL=1
MOVL C00494 V=30.0 PL=1
MOVL C00495 V=30.0 PL=1
MOVL C00496 V=30.0 PL=1
MOVL C00497 V=30.0 PL=1
MOVL C00498 V=30.0 PL=1
MOVL C00499 V=30.0 PL=1
MOVL C00500 V=30.0 PL=1
MOVL C00501 V=30.0 PL=1
MOVL C00502 V=30.0 PL=1
MOVL C00503 V=30.0 PL=1
MOVL C00504 V=30.0 PL=1
MOVL C00505 V=30.0 PL=1
MOVL C00506 V=30.0 PL=1
MOVL C00507 V=30.0 PL=1
MOVL C00508 V=30.0 PL=1
MOVL C00509 V=30.0 PL=1
MOVL C00510 V=30.0 PL=1
MOVL C00511 V=30.0 PL=1
MOVL C00512 V=30.0 PL=1
MOVL C00513 V=30.0 PL=1
MOVL C00514 V=30.0 PL=1
MOVL C00515 V=30.0 PL=1
MOVL C00516 V=30.0 PL=1
MOVL C00517 V=30.0 PL=1
MOVL C00518 V=30.0 PL=1
MOVL C00519 V=30.0 PL=1
MOVL C00520 V=30.0 PL=1
MOVL C00521 V=30.0 PL=1
MOVL C00522 V=30.0 PL=1
MOVL C00523 V=30.0 PL=1
MOVL C00524 V=30.0 PL=1
MOVL C00525 V=30.0 PL=1
MOVL C00526 V=30.0 PL=1
MOVL C00527 V=30.0 PL=1
MOVL C00528 V=30.0 PL=1
MOVL C00529 V=30.0 PL=1
MOVL C00530 V=30.0 PL=1
MOVL C00531 V=30.0 PL=1
MOVL C00532 V=30.0 PL=1
MOVL C00533 V=30.0 PL=1
MOVL C00534 V=30.0 PL=1
MOVL C00535 V=30.0 PL=1
MOVL C00536 V=30.0 PL=1
MOVL C00537 V=30.0 PL=1
MOVL C00538 V=30.0 PL=1
MOVL C00539 V=30.0 PL=1
MOVL C00540 V=30.0 PL=1
MOVL C00541 V=30.0 PL=1
MOVL C00542 V=30.0 PL=1
MOVL C00543 V=30.0 PL=1
MOVL C00544 V=30.0 PL=1
MOVL C00545 V=130.0 PL=1
MOVL C00546 V=130.0 PL=1
MOVL C00547 V=60.0 PL=1
MOVL C00548 V=60.0 PL=1
MOVL C00549 V=60.0 PL=1
MOVL C00550 V=60.0 PL=1
MOVL C00551 V=130.0 PL=1
MOVL C00552 V=30.0 PL=1
MOVL C00553 V=30.0 PL=1
MOVL C00554 V=30.0 PL=1
MOVL C00555 V=30.0 PL=1
MOVL C00556 V=30.0 PL=1
MOVL C00557 V=30.0 PL=1
MOVL C00558 V=30.0 PL=1
MOVL C00559 V=30.0 PL=1
MOVL C00560 V=130.0 PL=1
MOVL C00561 V=130.0 PL=1
MOVL C00562 V=30.0 PL=1
MOVL C00563 V=130.0 PL=1
MOVL C00564 V=30.0 PL=1
MOVL C00565 V=130.0 PL=1
MOVL C00566 V=30.0 PL=1
MOVL C00567 V=130.0 PL=1
MOVL C00568 V=20.0 PL=1
MOVL C00569 V=130.0 PL=1
MOVL C00570 V=30.0 PL=1
MOVL C00571 V=30.0 PL=1
MOVL C00572 V=30.0 PL=1
MOVL C00573 V=30.0 PL=1
MOVL C00574 V=30.0 PL=1
MOVL C00575 V=30.0 PL=1
MOVL C00576 V=30.0 PL=1
MOVL C00577 V=30.0 PL=1
MOVL C00578 V=30.0 PL=1
MOVL C00579 V=30.0 PL=1
MOVL C00580 V=30.0 PL=1
MOVL C00581 V=30.0 PL=1
MOVL C00582 V=30.0 PL=1
MOVL C00583 V=30.0 PL=1
MOVL C00584 V=30.0 PL=1
MOVL C00585 V=30.0 PL=1
MOVL C00586 V=30.0 PL=1
MOVL C00587 V=30.0 PL=1
MOVL C00588 V=30.0 PL=1
MOVL C00589 V=30.0 PL=1
MOVL C00590 V=30.0 PL=1
MOVL C00591 V=30.0 PL=1
MOVL C00592 V=30.0 PL=1
MOVL C00593 V=30.0 PL=1
MOVL C00594 V=30.0 PL=1
MOVL C00595 V=30.0 PL=1
MOVL C00596 V=30.0 PL=1
MOVL C00597 V=30.0 PL=1
MOVL C00598 V=30.0 PL=1
MOVL C00599 V=30.0 PL=1
MOVL C00600 V=30.0 PL=1
MOVL C00601 V=30.0 PL=1
MOVL C00602 V=30.0 PL=1
MOVL C00603 V=30.0 PL=1
MOVL C00604 V=30.0 PL=1
MOVL C00605 V=30.0 PL=1
MOVL C00606 V=30.0 PL=1
MOVL C00607 V=30.0 PL=1
MOVL C00608 V=30.0 PL=1
MOVL C00609 V=30.0 PL=1
MOVL C00610 V=30.0 PL=1
MOVL C00611 V=30.0 PL=1
MOVL C00612 V=30.0 PL=1
MOVL C00613 V=30.0 PL=1
MOVL C00614 V=30.0 PL=1
MOVL C00615 V=30.0 PL=1
MOVL C00616 V=30.0 PL=1
MOVL C00617 V=30.0 PL=1
MOVL C00618 V=30.0 PL=1
MOVL C00619 V=30.0 PL=1
MOVL C00620 V=30.0 PL=1
MOVL C00621 V=30.0 PL=1
MOVL C00622 V=30.0 PL=1
MOVL C00623 V=30.0 PL=1
MOVL C00624 V=30.0 PL=1
MOVL C00625 V=30.0 PL=1
MOVL C00626 V=30.0 PL=1
MOVL C00627 V=30.0 PL=1
MOVL C00628 V=30.0 PL=1
MOVL C00629 V=30.0 PL=1
MOVL C00630 V=30.0 PL=1
MOVL C00631 V=30.0 PL=1
MOVL C00632 V=30.0 PL=1
MOVL C00633 V=30.0 PL=1
MOVL C00634 V=30.0 PL=1
MOVL C00635 V=30.0 PL=1
MOVL C00636 V=30.0 PL=1
MOVL C00637 V=30.0 PL=1
MOVL C00638 V=30.0 PL=1
MOVL C00639 V=30.0 PL=1
MOVL C00640 V=30.0 PL=1
MOVL C00641 V=30.0 PL=1
MOVL C00642 V=30.0 PL=1
MOVL C00643 V=30.0 PL=1
MOVL C00644 V=30.0 PL=1
MOVL C00645 V=30.0 PL=1
MOVL C00646 V=130.0 PL=1
MOVL C00647 V=130.0 PL=1
MOVL C00648 V=30.0 PL=1
MOVL C00649 V=30.0 PL=1
MOVL C00650 V=30.0 PL=1
MOVL C00651 V=30.0 PL=1
MOVL C00652 V=30.0 PL=1
MOVL C00653 V=30.0 PL=1
MOVL C00654 V=30.0 PL=1
MOVL C00655 V=30.0 PL=1
MOVL C00656 V=30.0 PL=1
MOVL C00657 V=30.0 PL=1
MOVL C00658 V=30.0 PL=1
MOVL C00659 V=30.0 PL=1
MOVL C00660 V=30.0 PL=1
MOVL C00661 V=30.0 PL=1
MOVL C00662 V=30.0 PL=1
MOVL C00663 V=30.0 PL=1
MOVL C00664 V=30.0 PL=1
MOVL C00665 V=30.0 PL=1
MOVL C00666 V=30.0 PL=1
MOVL C00667 V=30.0 PL=1
MOVL C00668 V=30.0 PL=1
MOVL C00669 V=30.0 PL=1
MOVL C00670 V=30.0 PL=1
MOVL C00671 V=30.0 PL=1
MOVL C00672 V=30.0 PL=1
MOVL C00673 V=30.0 PL=1
MOVL C00674 V=30.0 PL=1
MOVL C00675 V=30.0 PL=1
MOVL C00676 V=30.0 PL=1
MOVL C00677 V=30.0 PL=1
MOVL C00678 V=30.0 PL=1
MOVL C00679 V=30.0 PL=1
MOVL C00680 V=30.0 PL=1
MOVL C00681 V=30.0 PL=1
MOVL C00682 V=30.0 PL=1
MOVL C00683 V=30.0 PL=1
MOVL C00684 V=30.0 PL=1
MOVL C00685 V=30.0 PL=1
MOVL C00686 V=30.0 PL=1
MOVL C00687 V=30.0 PL=1
MOVL C00688 V=30.0 PL=1
MOVL C00689 V=30.0 PL=1
MOVL C00690 V=30.0 PL=1
MOVL C00691 V=30.0 PL=1
MOVL C00692 V=30.0 PL=1
MOVL C00693 V=30.0 PL=1
MOVL C00694 V=30.0 PL=1
MOVL C00695 V=30.0 PL=1
MOVL C00696 V=30.0 PL=1
MOVL C00697 V=30.0 PL=1
MOVL C00698 V=30.0 PL=1
MOVL C00699 V=30.0 PL=1
MOVL C00700 V=30.0 PL=1
MOVL C00701 V=30.0 PL=1
MOVL C00702 V=30.0 PL=1
MOVL C00703 V=30.0 PL=1
MOVL C00704 V=30.0 PL=1
MOVL C00705 V=30.0 PL=1
MOVL C00706 V=30.0 PL=1
MOVL C00707 V=30.0 PL=1
MOVL C00708 V=30.0 PL=1
MOVL C00709 V=30.0 PL=1
MOVL C00710 V=30.0 PL=1
MOVL C00711 V=30.0 PL=1
MOVL C00712 V=30.0 PL=1
MOVL C00713 V=30.0 PL=1
MOVL C00714 V=30.0 PL=1
MOVL C00715 V=30.0 PL=1
MOVL C00716 V=30.0 PL=1
MOVL C00717 V=30.0 PL=1
MOVL C00718 V=30.0 PL=1
MOVL C00719 V=30.0 PL=1
MOVL C00720 V=30.0 PL=1
MOVL C00721 V=30.0 PL=1
MOVL C00722 V=30.0 PL=1
MOVL C00723 V=30.0 PL=1
MOVL C00724 V=30.0 PL=1
MOVL C00725 V=30.0 PL=1
MOVL C00726 V=30.0 PL=1
MOVL C00727 V=30.0 PL=1
MOVL C00728 V=130.0 PL=1
MOVL C00729 V=130.0 PL=1
MOVL C00730 V=30.0 PL=1
MOVL C00731 V=130.0 PL=1
MOVL C00732 V=30.0 PL=1
MOVL C00733 V=30.0 PL=1
MOVL C00734 V=30.0 PL=1
MOVL C00735 V=30.0 PL=1
MOVL C00736 V=30.0 PL=1
MOVL C00737 V=30.0 PL=1
MOVL C00738 V=30.0 PL=1
MOVL C00739 V=30.0 PL=1
MOVL C00740 V=30.0 PL=1
MOVL C00741 V=30.0 PL=1
MOVL C00742 V=30.0 PL=1
MOVL C00743 V=30.0 PL=1
MOVL C00744 V=30.0 PL=1
MOVL C00745 V=30.0 PL=1
MOVL C00746 V=30.0 PL=1
MOVL C00747 V=30.0 PL=1
MOVL C00748 V=30.0 PL=1
MOVL C00749 V=30.0 PL=1
MOVL C00750 V=30.0 PL=1
MOVL C00751 V=30.0 PL=1
MOVL C00752 V=30.0 PL=1
MOVL C00753 V=30.0 PL=1
MOVL C00754 V=30.0 PL=1
MOVL C00755 V=30.0 PL=1
MOVL C00756 V=30.0 PL=1
MOVL C00757 V=30.0 PL=1
MOVL C00758 V=30.0 PL=1
MOVL C00759 V=30.0 PL=1
MOVL C00760 V=30.0 PL=1
MOVL C00761 V=30.0 PL=1
MOVL C00762 V=30.0 PL=1
MOVL C00763 V=30.0 PL=1
MOVL C00764 V=30.0 PL=1
MOVL C00765 V=30.0 PL=1
MOVL C00766 V=30.0 PL=1
MOVL C00767 V=30.0 PL=1
MOVL C00768 V=30.0 PL=1
MOVL C00769 V=30.0 PL=1
MOVL C00770 V=30.0 PL=1
MOVL C00771 V=30.0 PL=1
MOVL C00772 V=30.0 PL=1
MOVL C00773 V=30.0 PL=1
MOVL C00774 V=30.0 PL=1
MOVL C00775 V=30.0 PL=1
MOVL C00776 V=30.0 PL=1
MOVL C00777 V=30.0 PL=1
MOVL C00778 V=30.0 PL=1
MOVL C00779 V=30.0 PL=1
MOVL C00780 V=30.0 PL=1
MOVL C00781 V=30.0 PL=1
MOVL C00782 V=30.0 PL=1
MOVL C00783 V=30.0 PL=1
MOVL C00784 V=30.0 PL=1
MOVL C00785 V=30.0 PL=1
MOVL C00786 V=30.0 PL=1
MOVL C00787 V=30.0 PL=1
MOVL C00788 V=30.0 PL=1
MOVL C00789 V=30.0 PL=1
MOVL C00790 V=30.0 PL=1
MOVL C00791 V=30.0 PL=1
MOVL C00792 V=30.0 PL=1
MOVL C00793 V=30.0 PL=1
MOVL C00794 V=30.0 PL=1
MOVL C00795 V=30.0 PL=1
MOVL C00796 V=30.0 PL=1
MOVL C00797 V=30.0 PL=1
MOVL C00798 V=30.0 PL=1
MOVL C00799 V=30.0 PL=1
MOVL C00800 V=30.0 PL=1
MOVL C00801 V=30.0 PL=1
MOVL C00802 V=30.0 PL=1
MOVL C00803 V=30.0 PL=1
MOVL C00804 V=30.0 PL=1
MOVL C00805 V=30.0 PL=1
MOVL C00806 V=30.0 PL=1
MOVL C00807 V=30.0 PL=1
MOVL C00808 V=30.0 PL=1
MOVL C00809 V=30.0 PL=1
MOVL C00810 V=30.0 PL=1
MOVL C00811 V=130.0 PL=1
MOVL C00812 V=130.0 PL=1
MOVL C00813 V=130.0 PL=1
MOVL C00814 V=30.0 PL=1
MOVL C00815 V=30.0 PL=1
MOVL C00816 V=30.0 PL=1
MOVL C00817 V=30.0 PL=1
MOVL C00818 V=30.0 PL=1
MOVL C00819 V=30.0 PL=1
MOVL C00820 V=30.0 PL=1
MOVL C00821 V=30.0 PL=1
MOVL C00822 V=30.0 PL=1
MOVL C00823 V=30.0 PL=1
MOVL C00824 V=30.0 PL=1
MOVL C00825 V=30.0 PL=1
MOVL C00826 V=30.0 PL=1
MOVL C00827 V=30.0 PL=1
MOVL C00828 V=30.0 PL=1
MOVL C00829 V=30.0 PL=1
MOVL C00830 V=30.0 PL=1
MOVL C00831 V=30.0 PL=1
MOVL C00832 V=30.0 PL=1
MOVL C00833 V=30.0 PL=1
MOVL C00834 V=30.0 PL=1
MOVL C00835 V=30.0 PL=1
MOVL C00836 V=30.0 PL=1
MOVL C00837 V=30.0 PL=1
MOVL C00838 V=30.0 PL=1
MOVL C00839 V=30.0 PL=1
MOVL C00840 V=30.0 PL=1
MOVL C00841 V=30.0 PL=1
MOVL C00842 V=30.0 PL=1
MOVL C00843 V=30.0 PL=1
MOVL C00844 V=30.0 PL=1
MOVL C00845 V=30.0 PL=1
MOVL C00846 V=30.0 PL=1
MOVL C00847 V=30.0 PL=1
MOVL C00848 V=30.0 PL=1
MOVL C00849 V=30.0 PL=1
MOVL C00850 V=30.0 PL=1
MOVL C00851 V=30.0 PL=1
MOVL C00852 V=30.0 PL=1
MOVL C00853 V=30.0 PL=1
MOVL C00854 V=30.0 PL=1
MOVL C00855 V=30.0 PL=1
MOVL C00856 V=30.0 PL=1
MOVL C00857 V=30.0 PL=1
MOVL C00858 V=30.0 PL=1
MOVL C00859 V=30.0 PL=1
MOVL C00860 V=30.0 PL=1
MOVL C00861 V=30.0 PL=1
MOVL C00862 V=30.0 PL=1
MOVL C00863 V=30.0 PL=1
MOVL C00864 V=30.0 PL=1
MOVL C00865 V=30.0 PL=1
MOVL C00866 V=30.0 PL=1
MOVL C00867 V=30.0 PL=1
MOVL C00868 V=30.0 PL=1
MOVL C00869 V=30.0 PL=1
MOVL C00870 V=30.0 PL=1
MOVL C00871 V=30.0 PL=1
MOVL C00872 V=30.0 PL=1
MOVL C00873 V=30.0 PL=1
MOVL C00874 V=30.0 PL=1
MOVL C00875 V=30.0 PL=1
MOVL C00876 V=30.0 PL=1
MOVL C00877 V=30.0 PL=1
MOVL C00878 V=30.0 PL=1
MOVL C00879 V=30.0 PL=1
MOVL C00880 V=30.0 PL=1
MOVL C00881 V=30.0 PL=1
MOVL C00882 V=30.0 PL=1
MOVL C00883 V=30.0 PL=1
MOVL C00884 V=30.0 PL=1
MOVL C00885 V=30.0 PL=1
MOVL C00886 V=30.0 PL=1
MOVL C00887 V=30.0 PL=1
MOVL C00888 V=30.0 PL=1
MOVL C00889 V=30.0 PL=1
MOVL C00890 V=30.0 PL=1
MOVL C00891 V=30.0 PL=1
MOVL C00892 V=30.0 PL=1
MOVL C00893 V=30.0 PL=1
MOVL C00894 V=30.0 PL=1
MOVL C00895 V=30.0 PL=1
MOVL C00896 V=130.0 PL=1
MOVL C00897 V=130.0 PL=1
MOVL C00898 V=60.0 PL=1
MOVL C00899 V=60.0 PL=1
MOVL C00900 V=60.0 PL=1
MOVL C00901 V=60.0 PL=1
MOVL C00902 V=130.0 PL=1
MOVL C00903 V=30.0 PL=1
MOVL C00904 V=30.0 PL=1
MOVL C00905 V=30.0 PL=1
MOVL C00906 V=30.0 PL=1
MOVL C00907 V=30.0 PL=1
MOVL C00908 V=30.0 PL=1
MOVL C00909 V=30.0 PL=1
MOVL C00910 V=30.0 PL=1
MOVL C00911 V=130.0 PL=1
MOVL C00912 V=130.0 PL=1
MOVL C00913 V=30.0 PL=1
MOVL C00914 V=130.0 PL=1
MOVL C00915 V=30.0 PL=1
MOVL C00916 V=130.0 PL=1
MOVL C00917 V=30.0 PL=1
MOVL C00918 V=130.0 PL=1
MOVL C00919 V=20.0 PL=1
MOVL C00920 V=130.0 PL=1
MOVL C00921 V=30.0 PL=1
MOVL C00922 V=30.0 PL=1
MOVL C00923 V=30.0 PL=1
MOVL C00924 V=30.0 PL=1
MOVL C00925 V=30.0 PL=1
MOVL C00926 V=30.0 PL=1
MOVL C00927 V=30.0 PL=1
MOVL C00928 V=30.0 PL=1
MOVL C00929 V=30.0 PL=1
MOVL C00930 V=30.0 PL=1
MOVL C00931 V=30.0 PL=1
MOVL C00932 V=30.0 PL=1
MOVL C00933 V=30.0 PL=1
MOVL C00934 V=30.0 PL=1
MOVL C00935 V=30.0 PL=1
MOVL C00936 V=30.0 PL=1
MOVL C00937 V=30.0 PL=1
MOVL C00938 V=30.0 PL=1
MOVL C00939 V=30.0 PL=1
MOVL C00940 V=30.0 PL=1
MOVL C00941 V=30.0 PL=1
MOVL C00942 V=30.0 PL=1
MOVL C00943 V=30.0 PL=1
MOVL C00944 V=30.0 PL=1
MOVL C00945 V=30.0 PL=1
MOVL C00946 V=30.0 PL=1
MOVL C00947 V=30.0 PL=1
MOVL C00948 V=30.0 PL=1
MOVL C00949 V=30.0 PL=1
MOVL C00950 V=30.0 PL=1
MOVL C00951 V=30.0 PL=1
MOVL C00952 V=30.0 PL=1
MOVL C00953 V=30.0 PL=1
MOVL C00954 V=30.0 PL=1
MOVL C00955 V=30.0 PL=1
MOVL C00956 V=30.0 PL=1
MOVL C00957 V=30.0 PL=1
MOVL C00958 V=30.0 PL=1
MOVL C00959 V=30.0 PL=1
MOVL C00960 V=30.0 PL=1
MOVL C00961 V=30.0 PL=1
MOVL C00962 V=30.0 PL=1
MOVL C00963 V=30.0 PL=1
MOVL C00964 V=30.0 PL=1
MOVL C00965 V=30.0 PL=1
MOVL C00966 V=30.0 PL=1
MOVL C00967 V=30.0 PL=1
MOVL C00968 V=30.0 PL=1
MOVL C00969 V=30.0 PL=1
MOVL C00970 V=30.0 PL=1
MOVL C00971 V=30.0 PL=1
MOVL C00972 V=30.0 PL=1
MOVL C00973 V=30.0 PL=1
MOVL C00974 V=30.0 PL=1
MOVL C00975 V=30.0 PL=1
MOVL C00976 V=30.0 PL=1
MOVL C00977 V=30.0 PL=1
MOVL C00978 V=30.0 PL=1
MOVL C00979 V=30.0 PL=1
MOVL C00980 V=30.0 PL=1
MOVL C00981 V=30.0 PL=1
MOVL C00982 V=30.0 PL=1
MOVL C00983 V=30.0 PL=1
MOVL C00984 V=30.0 PL=1
MOVL C00985 V=30.0 PL=1
MOVL C00986 V=30.0 PL=1
MOVL C00987 V=30.0 PL=1
MOVL C00988 V=30.0 PL=1
MOVL C00989 V=30.0 PL=1
END
